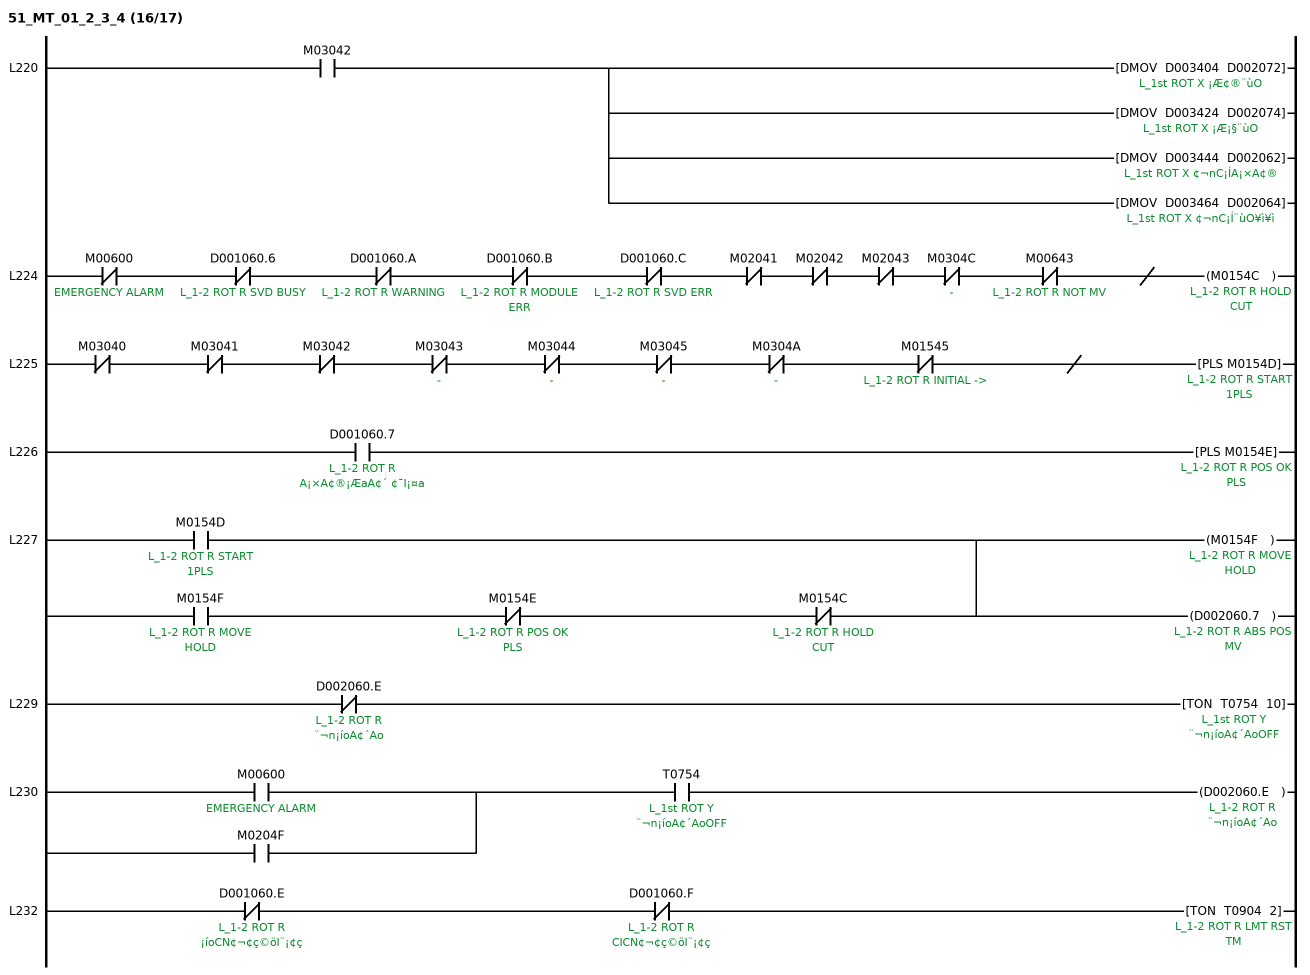
[picture p264: 51_MT_01_2_3_4 rungs L220-L232]
; L220
LOAD      M03042
DMOV      D003404 D002072	// L_1st ROT X ¡Æ¢®¨ùO
DMOV      D003424 D002074	// L_1st ROT X ¡Æ¡§¨ùO
DMOV      D003444 D002062	// L_1st ROT X ¢¬nC¡ÍA¡×A¢®
DMOV      D003464 D002064	// L_1st ROT X ¢¬nC¡Í¨ùO¥ì¥ì
; L224
LOAD NOT  M00600	// EMERGENCY ALARM
AND NOT   D001060.6	// L_1-2 ROT R SVD BUSY
AND NOT   D001060.A	// L_1-2 ROT R WARNING
AND NOT   D001060.B	// L_1-2 ROT R MODULE ERR
AND NOT   D001060.C	// L_1-2 ROT R SVD ERR
AND NOT   M02041
AND NOT   M02042
AND NOT   M02043
AND NOT   M0304C	// -
AND NOT   M00643	// L_1-2 ROT R NOT MV
NOT
OUT       M0154C	// L_1-2 ROT R HOLD CUT
; L225
LOAD NOT  M03040
AND NOT   M03041
AND NOT   M03042
AND NOT   M03043	// -
AND NOT   M03044	// -
AND NOT   M03045	// -
AND NOT   M0304A	// -
AND NOT   M01545	// L_1-2 ROT R INITIAL ->
NOT
OUTP      M0154D	// L_1-2 ROT R START 1PLS
; L226
LOAD      D001060.7	// L_1-2 ROT R A¡×A¢®¡ÆaA¢´ ¢¯I¡¤a
OUTP      M0154E	// L_1-2 ROT R POS OK PLS
; L227
LOAD      M0154D	// L_1-2 ROT R START 1PLS
LOAD      M0154F	// L_1-2 ROT R MOVE HOLD
AND NOT   M0154E	// L_1-2 ROT R POS OK PLS
AND NOT   M0154C	// L_1-2 ROT R HOLD CUT
OR LOAD
OUT       M0154F	// L_1-2 ROT R MOVE HOLD
OUT       D002060.7	// L_1-2 ROT R ABS POS MV
; L229
LOAD NOT  D002060.E	// L_1-2 ROT R ¨¬n¡íoA¢´Ao
TON       T0754 10	// L_1st ROT Y ¨¬n¡íoA¢´AoOFF
; L230
LOAD      M00600	// EMERGENCY ALARM
OR        M0204F
AND       T0754	// L_1st ROT Y ¨¬n¡íoA¢´AoOFF
OUT       D002060.E	// L_1-2 ROT R ¨¬n¡íoA¢´Ao
; L232
LOAD NOT  D001060.E	// L_1-2 ROT R ¡íoCN¢¬¢ç©öI¨¡¢ç
AND NOT   D001060.F	// L_1-2 ROT R CICN¢¬¢ç©öI¨¡¢ç
TON       T0904 2	// L_1-2 ROT R LMT RST TM

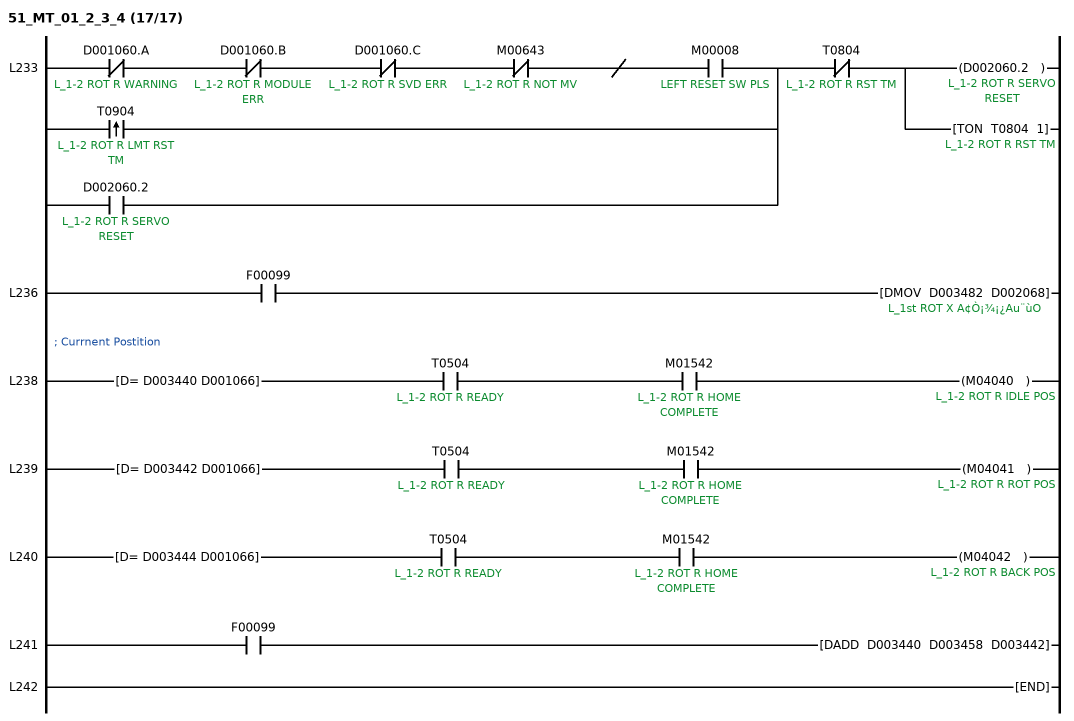
; L233
LOAD NOT  D001060.A	// L_1-2 ROT R WARNING
AND NOT   D001060.B	// L_1-2 ROT R MODULE ERR
AND NOT   D001060.C	// L_1-2 ROT R SVD ERR
AND NOT   M00643	// L_1-2 ROT R NOT MV
NOT
AND       M00008	// LEFT RESET SW PLS
ORP       T0904	// L_1-2 ROT R LMT RST TM
OR        D002060.2	// L_1-2 ROT R SERVO RESET
AND NOT   T0804	// L_1-2 ROT R RST TM
OUT       D002060.2	// L_1-2 ROT R SERVO RESET
TON       T0804 1	// L_1-2 ROT R RST TM
; L236
LOAD      F00099
DMOV      D003482 D002068	// L_1st ROT X A¢Ò¡¾¡¿Au¨ùO
// Currnent Postition
; L238
LOADD=    D003440 D001066
AND       T0504	// L_1-2 ROT R READY
AND       M01542	// L_1-2 ROT R HOME COMPLETE
OUT       M04040	// L_1-2 ROT R IDLE POS
; L239
LOADD=    D003442 D001066
AND       T0504	// L_1-2 ROT R READY
AND       M01542	// L_1-2 ROT R HOME COMPLETE
OUT       M04041	// L_1-2 ROT R ROT POS
; L240
LOADD=    D003444 D001066
AND       T0504	// L_1-2 ROT R READY
AND       M01542	// L_1-2 ROT R HOME COMPLETE
OUT       M04042	// L_1-2 ROT R BACK POS
; L241
LOAD      F00099
DADD      D003440 D003458 D003442
; L242
END

PROGRAM 52_MT_05_6_7_8 (task: ¨ö¨¬A¥ì CA¡¤I¡¾¡¿¡¤¡Í)

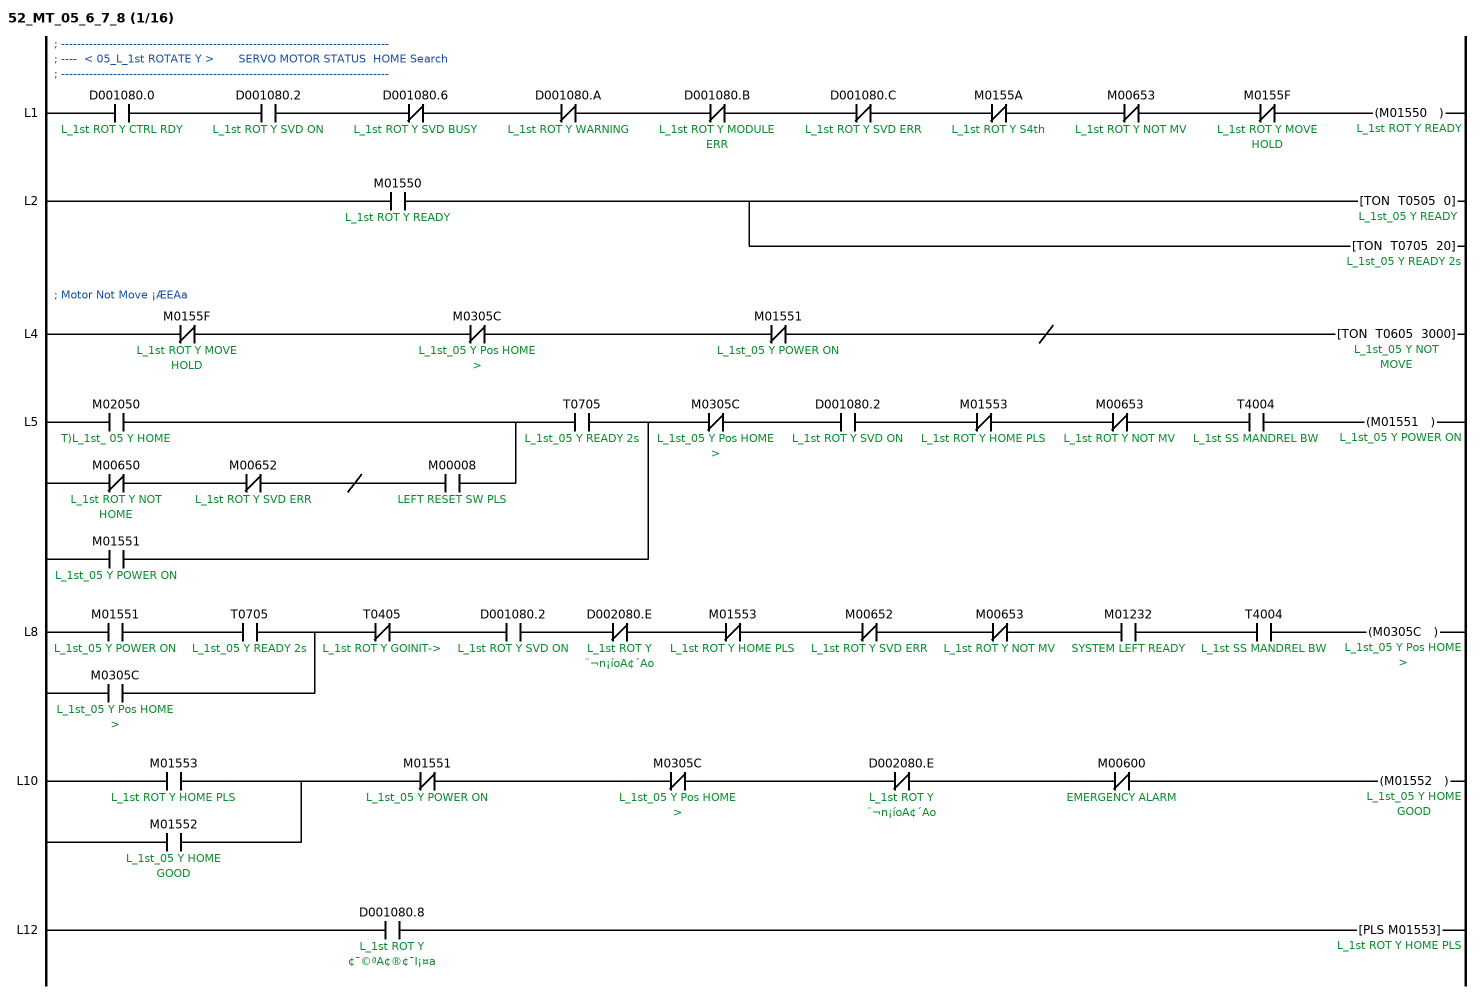
// ----------------------------------------------------------------------------------
// 
// ----  < 05_L_1st ROTATE Y >       SERVO MOTOR STATUS  HOME Search
// 
// ----------------------------------------------------------------------------------
; L1
LOAD      D001080.0	// L_1st ROT Y CTRL RDY
AND       D001080.2	// L_1st ROT Y SVD ON
AND NOT   D001080.6	// L_1st ROT Y SVD BUSY
AND NOT   D001080.A	// L_1st ROT Y WARNING
AND NOT   D001080.B	// L_1st ROT Y MODULE ERR
AND NOT   D001080.C	// L_1st ROT Y SVD ERR
AND NOT   M0155A	// L_1st ROT Y S4th
AND NOT   M00653	// L_1st ROT Y NOT MV
AND NOT   M0155F	// L_1st ROT Y MOVE HOLD
OUT       M01550	// L_1st ROT Y READY
; L2
LOAD      M01550	// L_1st ROT Y READY
TON       T0505 0	// L_1st_05 Y READY
TON       T0705 20	// L_1st_05 Y READY 2s
; L4
LOAD NOT  M0155F	// L_1st ROT Y MOVE HOLD
AND NOT   M0305C	// L_1st_05 Y Pos HOME >
AND NOT   M01551	// L_1st_05 Y POWER ON
NOT
TON       T0605 3000	// L_1st_05 Y NOT MOVE
// output comment: Motor Not Move ¡ÆEAa
; L5
LOAD      M02050	// T)L_1st_ 05 Y HOME
LOAD NOT  M00650	// L_1st ROT Y NOT HOME
AND NOT   M00652	// L_1st ROT Y SVD ERR
NOT
AND       M00008	// LEFT RESET SW PLS
OR LOAD
AND       T0705	// L_1st_05 Y READY 2s
OR        M01551	// L_1st_05 Y POWER ON
AND NOT   M0305C	// L_1st_05 Y Pos HOME >
AND       D001080.2	// L_1st ROT Y SVD ON
AND NOT   M01553	// L_1st ROT Y HOME PLS
AND NOT   M00653	// L_1st ROT Y NOT MV
AND       T4004	// L_1st SS MANDREL BW
OUT       M01551	// L_1st_05 Y POWER ON
; L8
LOAD      M01551	// L_1st_05 Y POWER ON
AND       T0705	// L_1st_05 Y READY 2s
OR        M0305C	// L_1st_05 Y Pos HOME >
AND NOT   T0405	// L_1st ROT Y GOINIT->
AND       D001080.2	// L_1st ROT Y SVD ON
AND NOT   D002080.E	// L_1st ROT Y ¨¬n¡íoA¢´Ao
AND NOT   M01553	// L_1st ROT Y HOME PLS
AND NOT   M00652	// L_1st ROT Y SVD ERR
AND NOT   M00653	// L_1st ROT Y NOT MV
AND       M01232	// SYSTEM LEFT READY
AND       T4004	// L_1st SS MANDREL BW
OUT       M0305C	// L_1st_05 Y Pos HOME >
; L10
LOAD      M01553	// L_1st ROT Y HOME PLS
OR        M01552	// L_1st_05 Y HOME GOOD
AND NOT   M01551	// L_1st_05 Y POWER ON
AND NOT   M0305C	// L_1st_05 Y Pos HOME >
AND NOT   D002080.E	// L_1st ROT Y ¨¬n¡íoA¢´Ao
AND NOT   M00600	// EMERGENCY ALARM
OUT       M01552	// L_1st_05 Y HOME GOOD
; L12
LOAD      D001080.8	// L_1st ROT Y ¢¯©ªA¢®¢¯I¡¤a
OUTP      M01553	// L_1st ROT Y HOME PLS

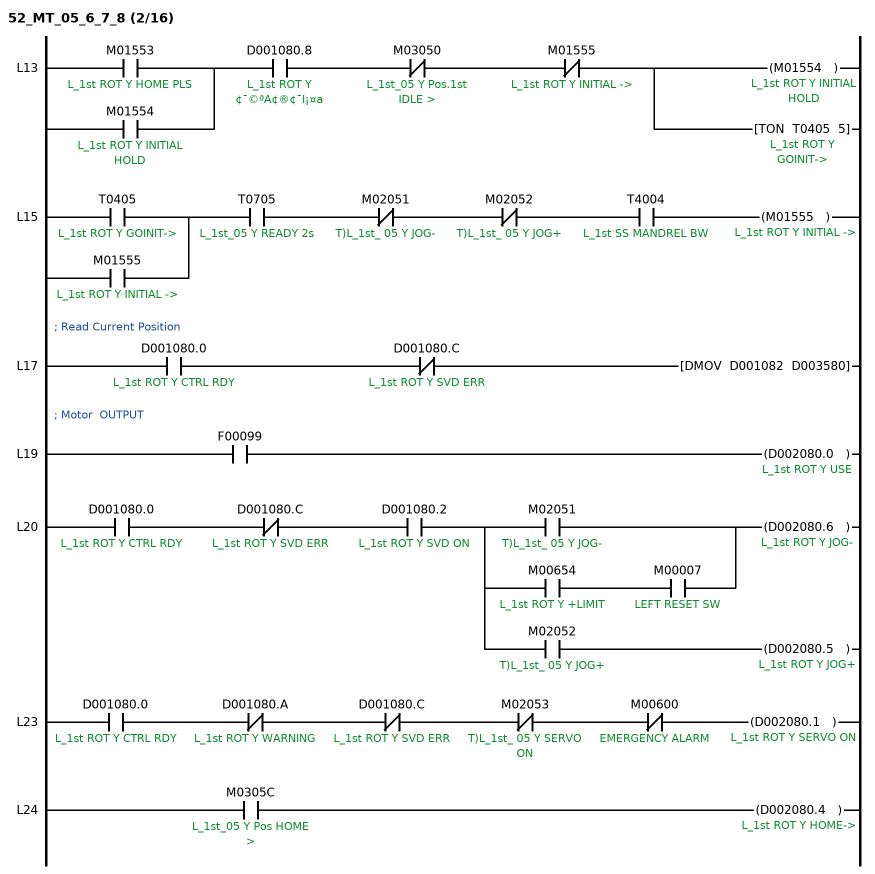
; L13
LOAD      M01553	// L_1st ROT Y HOME PLS
OR        M01554	// L_1st ROT Y INITIAL HOLD
AND       D001080.8	// L_1st ROT Y ¢¯©ªA¢®¢¯I¡¤a
AND NOT   M03050	// L_1st_05 Y Pos.1st IDLE >
AND NOT   M01555	// L_1st ROT Y INITIAL ->
OUT       M01554	// L_1st ROT Y INITIAL HOLD
TON       T0405 5	// L_1st ROT Y GOINIT->
; L15
LOAD      T0405	// L_1st ROT Y GOINIT->
OR        M01555	// L_1st ROT Y INITIAL ->
AND       T0705	// L_1st_05 Y READY 2s
AND NOT   M02051	// T)L_1st_ 05 Y JOG-
AND NOT   M02052	// T)L_1st_ 05 Y JOG+
AND       T4004	// L_1st SS MANDREL BW
OUT       M01555	// L_1st ROT Y INITIAL ->
; L17
LOAD      D001080.0	// L_1st ROT Y CTRL RDY
AND NOT   D001080.C	// L_1st ROT Y SVD ERR
DMOV      D001082 D003580
// output comment: Read Current Position
//  Motor  OUTPUT
; L19
LOAD      F00099
OUT       D002080.0	// L_1st ROT Y USE
; L20
LOAD      D001080.0	// L_1st ROT Y CTRL RDY
AND NOT   D001080.C	// L_1st ROT Y SVD ERR
AND       D001080.2	// L_1st ROT Y SVD ON
MPUSH
LOAD      M02051	// T)L_1st_ 05 Y JOG-
LOAD      M00654	// L_1st ROT Y +LIMIT
AND       M00007	// LEFT RESET SW
OR LOAD
AND LOAD
OUT       D002080.6	// L_1st ROT Y JOG-
MPOP
AND       M02052	// T)L_1st_ 05 Y JOG+
OUT       D002080.5	// L_1st ROT Y JOG+
; L23
LOAD      D001080.0	// L_1st ROT Y CTRL RDY
AND NOT   D001080.A	// L_1st ROT Y WARNING
AND NOT   D001080.C	// L_1st ROT Y SVD ERR
AND NOT   M02053	// T)L_1st_ 05 Y SERVO ON
AND NOT   M00600	// EMERGENCY ALARM
OUT       D002080.1	// L_1st ROT Y SERVO ON
; L24
LOAD      M0305C	// L_1st_05 Y Pos HOME >
OUT       D002080.4	// L_1st ROT Y HOME->

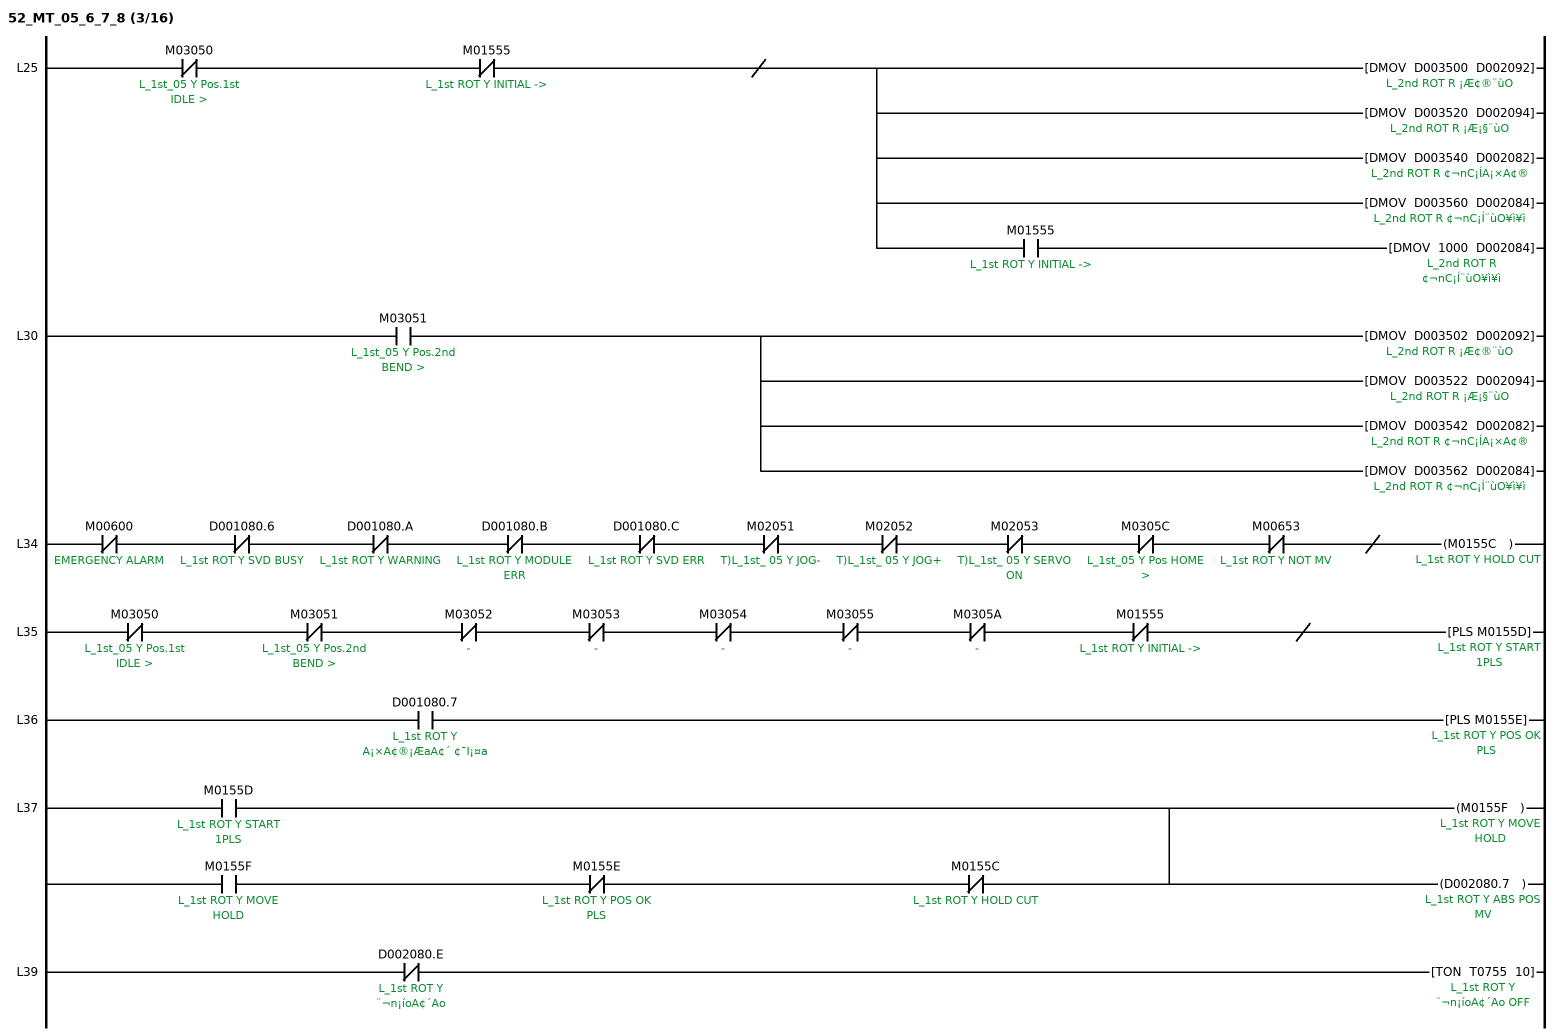
; L25
LOAD NOT  M03050	// L_1st_05 Y Pos.1st IDLE >
AND NOT   M01555	// L_1st ROT Y INITIAL ->
NOT
DMOV      D003500 D002092	// L_2nd ROT R ¡Æ¢®¨ùO
DMOV      D003520 D002094	// L_2nd ROT R ¡Æ¡§¨ùO
DMOV      D003540 D002082	// L_2nd ROT R ¢¬nC¡ÍA¡×A¢®
DMOV      D003560 D002084	// L_2nd ROT R ¢¬nC¡Í¨ùO¥ì¥ì
AND       M01555	// L_1st ROT Y INITIAL ->
DMOV      1000 D002084	// L_2nd ROT R ¢¬nC¡Í¨ùO¥ì¥ì
; L30
LOAD      M03051	// L_1st_05 Y Pos.2nd BEND >
DMOV      D003502 D002092	// L_2nd ROT R ¡Æ¢®¨ùO
DMOV      D003522 D002094	// L_2nd ROT R ¡Æ¡§¨ùO
DMOV      D003542 D002082	// L_2nd ROT R ¢¬nC¡ÍA¡×A¢®
DMOV      D003562 D002084	// L_2nd ROT R ¢¬nC¡Í¨ùO¥ì¥ì
; L34
LOAD NOT  M00600	// EMERGENCY ALARM
AND NOT   D001080.6	// L_1st ROT Y SVD BUSY
AND NOT   D001080.A	// L_1st ROT Y WARNING
AND NOT   D001080.B	// L_1st ROT Y MODULE ERR
AND NOT   D001080.C	// L_1st ROT Y SVD ERR
AND NOT   M02051	// T)L_1st_ 05 Y JOG-
AND NOT   M02052	// T)L_1st_ 05 Y JOG+
AND NOT   M02053	// T)L_1st_ 05 Y SERVO ON
AND NOT   M0305C	// L_1st_05 Y Pos HOME >
AND NOT   M00653	// L_1st ROT Y NOT MV
NOT
OUT       M0155C	// L_1st ROT Y HOLD CUT
; L35
LOAD NOT  M03050	// L_1st_05 Y Pos.1st IDLE >
AND NOT   M03051	// L_1st_05 Y Pos.2nd BEND >
AND NOT   M03052	// -
AND NOT   M03053	// -
AND NOT   M03054	// -
AND NOT   M03055	// -
AND NOT   M0305A	// -
AND NOT   M01555	// L_1st ROT Y INITIAL ->
NOT
OUTP      M0155D	// L_1st ROT Y START 1PLS
; L36
LOAD      D001080.7	// L_1st ROT Y A¡×A¢®¡ÆaA¢´ ¢¯I¡¤a
OUTP      M0155E	// L_1st ROT Y POS OK PLS
; L37
LOAD      M0155D	// L_1st ROT Y START 1PLS
LOAD      M0155F	// L_1st ROT Y MOVE HOLD
AND NOT   M0155E	// L_1st ROT Y POS OK PLS
AND NOT   M0155C	// L_1st ROT Y HOLD CUT
OR LOAD
OUT       M0155F	// L_1st ROT Y MOVE HOLD
OUT       D002080.7	// L_1st ROT Y ABS POS MV
; L39
LOAD NOT  D002080.E	// L_1st ROT Y ¨¬n¡íoA¢´Ao
TON       T0755 10	// L_1st ROT Y ¨¬n¡íoA¢´Ao OFF

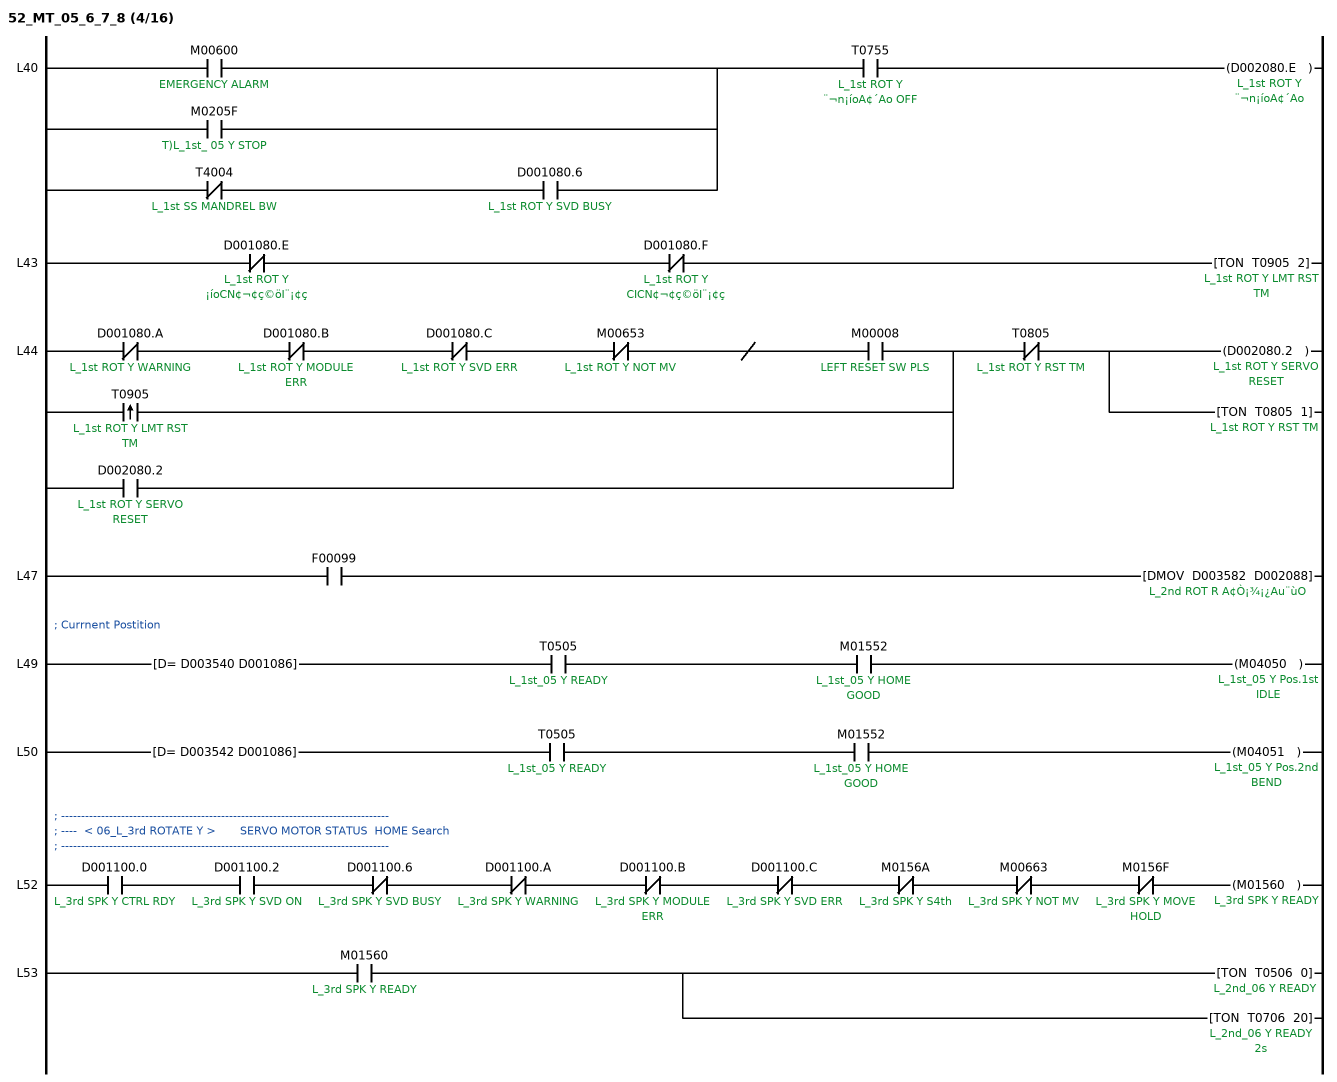
; L40
LOAD      M00600	// EMERGENCY ALARM
OR        M0205F	// T)L_1st_ 05 Y STOP
LOAD NOT  T4004	// L_1st SS MANDREL BW
AND       D001080.6	// L_1st ROT Y SVD BUSY
OR LOAD
AND       T0755	// L_1st ROT Y ¨¬n¡íoA¢´Ao OFF
OUT       D002080.E	// L_1st ROT Y ¨¬n¡íoA¢´Ao
; L43
LOAD NOT  D001080.E	// L_1st ROT Y ¡íoCN¢¬¢ç©öI¨¡¢ç
AND NOT   D001080.F	// L_1st ROT Y CICN¢¬¢ç©öI¨¡¢ç
TON       T0905 2	// L_1st ROT Y LMT RST TM
; L44
LOAD NOT  D001080.A	// L_1st ROT Y WARNING
AND NOT   D001080.B	// L_1st ROT Y MODULE ERR
AND NOT   D001080.C	// L_1st ROT Y SVD ERR
AND NOT   M00653	// L_1st ROT Y NOT MV
NOT
AND       M00008	// LEFT RESET SW PLS
ORP       T0905	// L_1st ROT Y LMT RST TM
OR        D002080.2	// L_1st ROT Y SERVO RESET
AND NOT   T0805	// L_1st ROT Y RST TM
OUT       D002080.2	// L_1st ROT Y SERVO RESET
TON       T0805 1	// L_1st ROT Y RST TM
; L47
LOAD      F00099
DMOV      D003582 D002088	// L_2nd ROT R A¢Ò¡¾¡¿Au¨ùO
// Currnent Postition
; L49
LOADD=    D003540 D001086
AND       T0505	// L_1st_05 Y READY
AND       M01552	// L_1st_05 Y HOME GOOD
OUT       M04050	// L_1st_05 Y Pos.1st IDLE
; L50
LOADD=    D003542 D001086
AND       T0505	// L_1st_05 Y READY
AND       M01552	// L_1st_05 Y HOME GOOD
OUT       M04051	// L_1st_05 Y Pos.2nd BEND
// ----------------------------------------------------------------------------------
// 
// ----  < 06_L_3rd ROTATE Y >       SERVO MOTOR STATUS  HOME Search
// 
// ----------------------------------------------------------------------------------
; L52
LOAD      D001100.0	// L_3rd SPK Y CTRL RDY
AND       D001100.2	// L_3rd SPK Y SVD ON
AND NOT   D001100.6	// L_3rd SPK Y SVD BUSY
AND NOT   D001100.A	// L_3rd SPK Y WARNING
AND NOT   D001100.B	// L_3rd SPK Y MODULE ERR
AND NOT   D001100.C	// L_3rd SPK Y SVD ERR
AND NOT   M0156A	// L_3rd SPK Y S4th
AND NOT   M00663	// L_3rd SPK Y NOT MV
AND NOT   M0156F	// L_3rd SPK Y MOVE HOLD
OUT       M01560	// L_3rd SPK Y READY
; L53
LOAD      M01560	// L_3rd SPK Y READY
TON       T0506 0	// L_2nd_06 Y READY
TON       T0706 20	// L_2nd_06 Y READY 2s

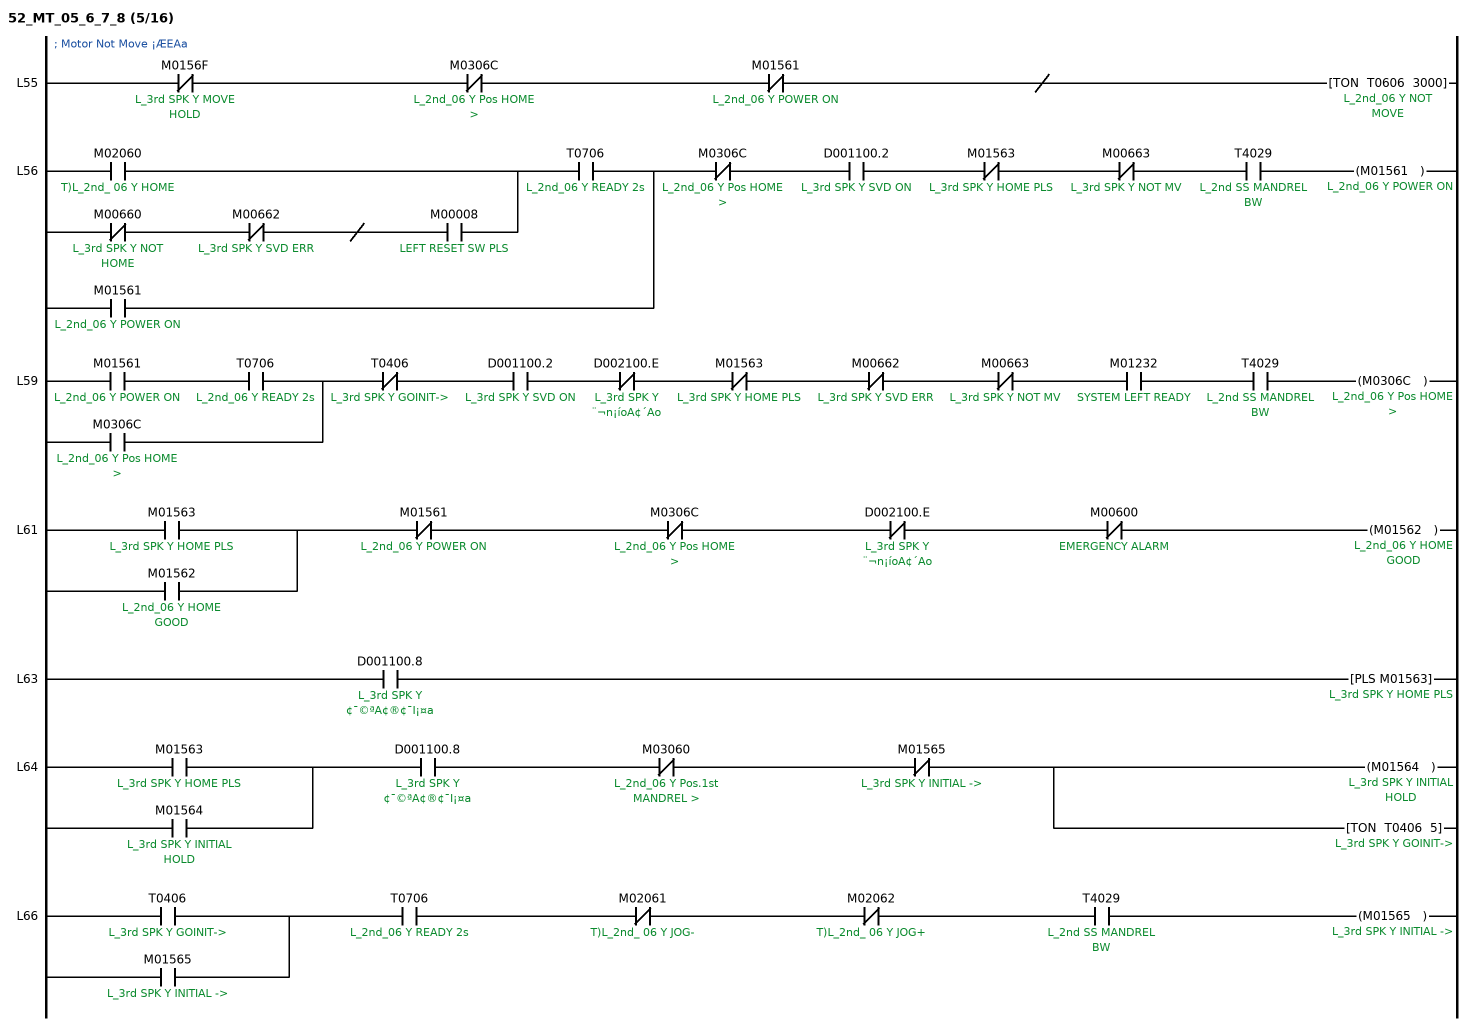
; L55
LOAD NOT  M0156F	// L_3rd SPK Y MOVE HOLD
AND NOT   M0306C	// L_2nd_06 Y Pos HOME >
AND NOT   M01561	// L_2nd_06 Y POWER ON
NOT
TON       T0606 3000	// L_2nd_06 Y NOT MOVE
// output comment: Motor Not Move ¡ÆEAa
; L56
LOAD      M02060	// T)L_2nd_ 06 Y HOME
LOAD NOT  M00660	// L_3rd SPK Y NOT HOME
AND NOT   M00662	// L_3rd SPK Y SVD ERR
NOT
AND       M00008	// LEFT RESET SW PLS
OR LOAD
AND       T0706	// L_2nd_06 Y READY 2s
OR        M01561	// L_2nd_06 Y POWER ON
AND NOT   M0306C	// L_2nd_06 Y Pos HOME >
AND       D001100.2	// L_3rd SPK Y SVD ON
AND NOT   M01563	// L_3rd SPK Y HOME PLS
AND NOT   M00663	// L_3rd SPK Y NOT MV
AND       T4029	// L_2nd SS MANDREL BW
OUT       M01561	// L_2nd_06 Y POWER ON
; L59
LOAD      M01561	// L_2nd_06 Y POWER ON
AND       T0706	// L_2nd_06 Y READY 2s
OR        M0306C	// L_2nd_06 Y Pos HOME >
AND NOT   T0406	// L_3rd SPK Y GOINIT->
AND       D001100.2	// L_3rd SPK Y SVD ON
AND NOT   D002100.E	// L_3rd SPK Y ¨¬n¡íoA¢´Ao
AND NOT   M01563	// L_3rd SPK Y HOME PLS
AND NOT   M00662	// L_3rd SPK Y SVD ERR
AND NOT   M00663	// L_3rd SPK Y NOT MV
AND       M01232	// SYSTEM LEFT READY
AND       T4029	// L_2nd SS MANDREL BW
OUT       M0306C	// L_2nd_06 Y Pos HOME >
; L61
LOAD      M01563	// L_3rd SPK Y HOME PLS
OR        M01562	// L_2nd_06 Y HOME GOOD
AND NOT   M01561	// L_2nd_06 Y POWER ON
AND NOT   M0306C	// L_2nd_06 Y Pos HOME >
AND NOT   D002100.E	// L_3rd SPK Y ¨¬n¡íoA¢´Ao
AND NOT   M00600	// EMERGENCY ALARM
OUT       M01562	// L_2nd_06 Y HOME GOOD
; L63
LOAD      D001100.8	// L_3rd SPK Y ¢¯©ªA¢®¢¯I¡¤a
OUTP      M01563	// L_3rd SPK Y HOME PLS
; L64
LOAD      M01563	// L_3rd SPK Y HOME PLS
OR        M01564	// L_3rd SPK Y INITIAL HOLD
AND       D001100.8	// L_3rd SPK Y ¢¯©ªA¢®¢¯I¡¤a
AND NOT   M03060	// L_2nd_06 Y Pos.1st MANDREL >
AND NOT   M01565	// L_3rd SPK Y INITIAL ->
OUT       M01564	// L_3rd SPK Y INITIAL HOLD
TON       T0406 5	// L_3rd SPK Y GOINIT->
; L66
LOAD      T0406	// L_3rd SPK Y GOINIT->
OR        M01565	// L_3rd SPK Y INITIAL ->
AND       T0706	// L_2nd_06 Y READY 2s
AND NOT   M02061	// T)L_2nd_ 06 Y JOG-
AND NOT   M02062	// T)L_2nd_ 06 Y JOG+
AND       T4029	// L_2nd SS MANDREL BW
OUT       M01565	// L_3rd SPK Y INITIAL ->

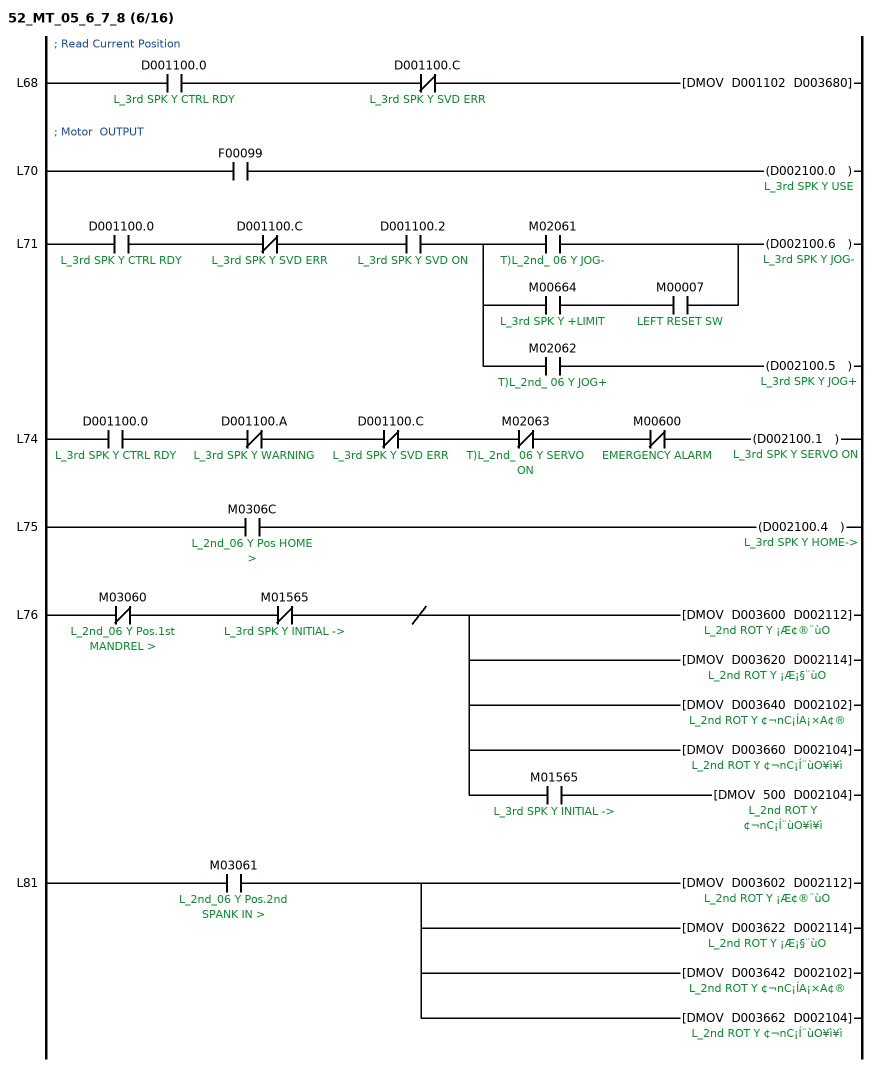
; L68
LOAD      D001100.0	// L_3rd SPK Y CTRL RDY
AND NOT   D001100.C	// L_3rd SPK Y SVD ERR
DMOV      D001102 D003680
// output comment: Read Current Position
//  Motor  OUTPUT
; L70
LOAD      F00099
OUT       D002100.0	// L_3rd SPK Y USE
; L71
LOAD      D001100.0	// L_3rd SPK Y CTRL RDY
AND NOT   D001100.C	// L_3rd SPK Y SVD ERR
AND       D001100.2	// L_3rd SPK Y SVD ON
MPUSH
LOAD      M02061	// T)L_2nd_ 06 Y JOG-
LOAD      M00664	// L_3rd SPK Y +LIMIT
AND       M00007	// LEFT RESET SW
OR LOAD
AND LOAD
OUT       D002100.6	// L_3rd SPK Y JOG-
MPOP
AND       M02062	// T)L_2nd_ 06 Y JOG+
OUT       D002100.5	// L_3rd SPK Y JOG+
; L74
LOAD      D001100.0	// L_3rd SPK Y CTRL RDY
AND NOT   D001100.A	// L_3rd SPK Y WARNING
AND NOT   D001100.C	// L_3rd SPK Y SVD ERR
AND NOT   M02063	// T)L_2nd_ 06 Y SERVO ON
AND NOT   M00600	// EMERGENCY ALARM
OUT       D002100.1	// L_3rd SPK Y SERVO ON
; L75
LOAD      M0306C	// L_2nd_06 Y Pos HOME >
OUT       D002100.4	// L_3rd SPK Y HOME->
; L76
LOAD NOT  M03060	// L_2nd_06 Y Pos.1st MANDREL >
AND NOT   M01565	// L_3rd SPK Y INITIAL ->
NOT
DMOV      D003600 D002112	// L_2nd ROT Y ¡Æ¢®¨ùO
DMOV      D003620 D002114	// L_2nd ROT Y ¡Æ¡§¨ùO
DMOV      D003640 D002102	// L_2nd ROT Y ¢¬nC¡ÍA¡×A¢®
DMOV      D003660 D002104	// L_2nd ROT Y ¢¬nC¡Í¨ùO¥ì¥ì
AND       M01565	// L_3rd SPK Y INITIAL ->
DMOV      500 D002104	// L_2nd ROT Y ¢¬nC¡Í¨ùO¥ì¥ì
; L81
LOAD      M03061	// L_2nd_06 Y Pos.2nd SPANK IN >
DMOV      D003602 D002112	// L_2nd ROT Y ¡Æ¢®¨ùO
DMOV      D003622 D002114	// L_2nd ROT Y ¡Æ¡§¨ùO
DMOV      D003642 D002102	// L_2nd ROT Y ¢¬nC¡ÍA¡×A¢®
DMOV      D003662 D002104	// L_2nd ROT Y ¢¬nC¡Í¨ùO¥ì¥ì

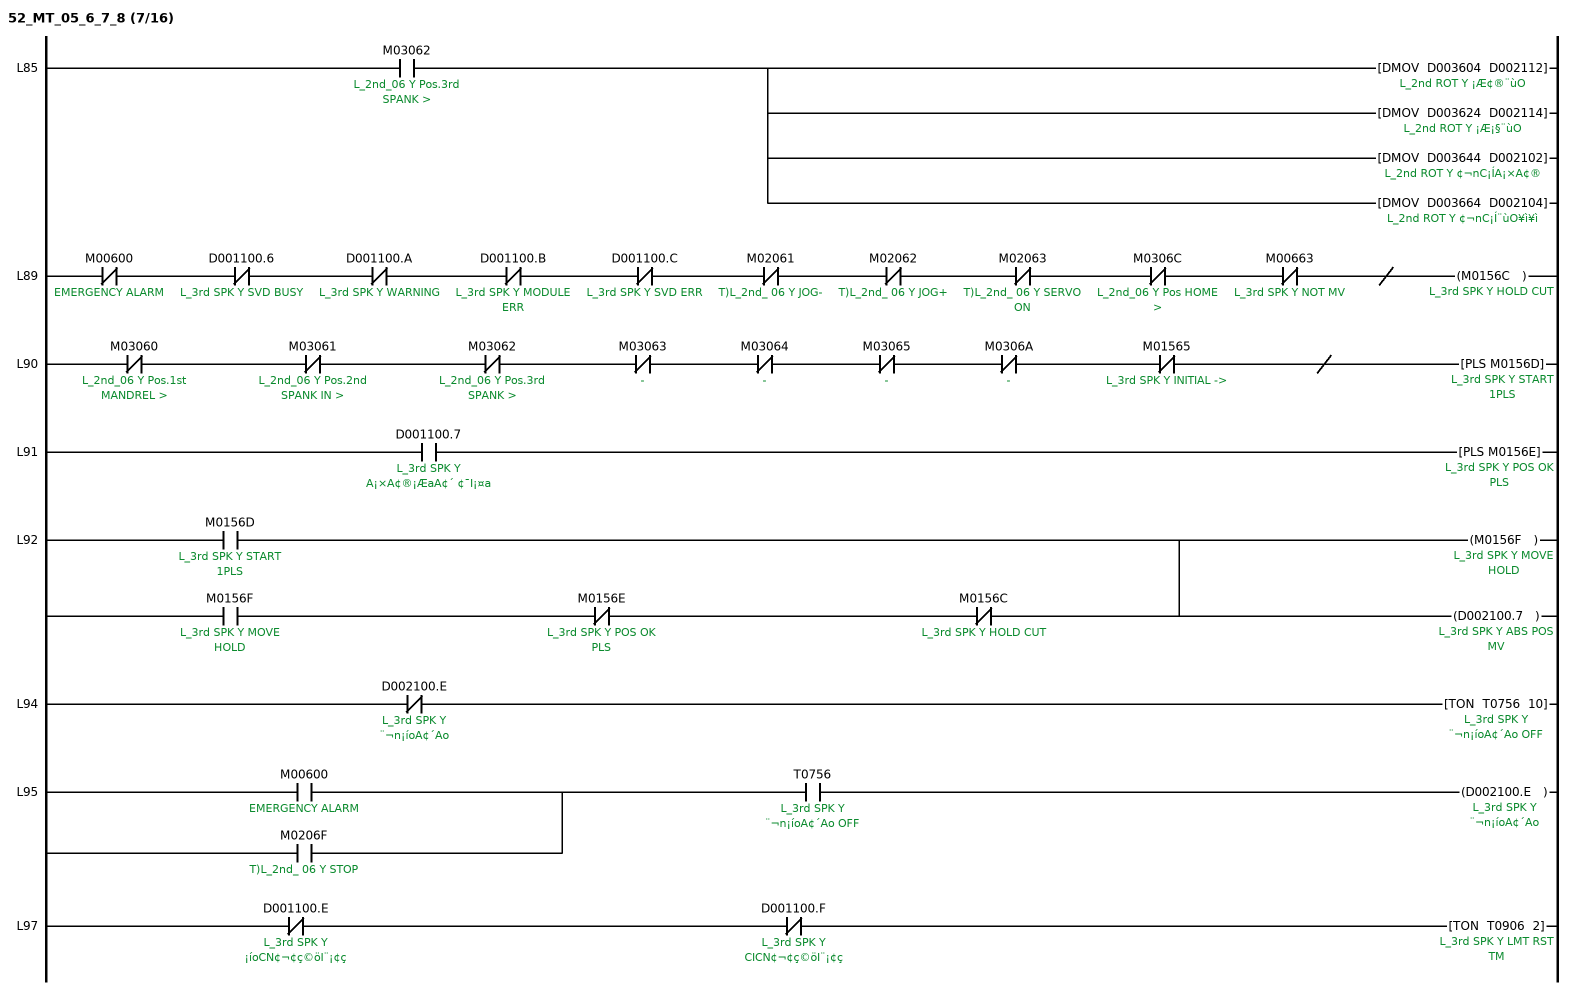
; L85
LOAD      M03062	// L_2nd_06 Y Pos.3rd SPANK >
DMOV      D003604 D002112	// L_2nd ROT Y ¡Æ¢®¨ùO
DMOV      D003624 D002114	// L_2nd ROT Y ¡Æ¡§¨ùO
DMOV      D003644 D002102	// L_2nd ROT Y ¢¬nC¡ÍA¡×A¢®
DMOV      D003664 D002104	// L_2nd ROT Y ¢¬nC¡Í¨ùO¥ì¥ì
; L89
LOAD NOT  M00600	// EMERGENCY ALARM
AND NOT   D001100.6	// L_3rd SPK Y SVD BUSY
AND NOT   D001100.A	// L_3rd SPK Y WARNING
AND NOT   D001100.B	// L_3rd SPK Y MODULE ERR
AND NOT   D001100.C	// L_3rd SPK Y SVD ERR
AND NOT   M02061	// T)L_2nd_ 06 Y JOG-
AND NOT   M02062	// T)L_2nd_ 06 Y JOG+
AND NOT   M02063	// T)L_2nd_ 06 Y SERVO ON
AND NOT   M0306C	// L_2nd_06 Y Pos HOME >
AND NOT   M00663	// L_3rd SPK Y NOT MV
NOT
OUT       M0156C	// L_3rd SPK Y HOLD CUT
; L90
LOAD NOT  M03060	// L_2nd_06 Y Pos.1st MANDREL >
AND NOT   M03061	// L_2nd_06 Y Pos.2nd SPANK IN >
AND NOT   M03062	// L_2nd_06 Y Pos.3rd SPANK >
AND NOT   M03063	// -
AND NOT   M03064	// -
AND NOT   M03065	// -
AND NOT   M0306A	// -
AND NOT   M01565	// L_3rd SPK Y INITIAL ->
NOT
OUTP      M0156D	// L_3rd SPK Y START 1PLS
; L91
LOAD      D001100.7	// L_3rd SPK Y A¡×A¢®¡ÆaA¢´ ¢¯I¡¤a
OUTP      M0156E	// L_3rd SPK Y POS OK PLS
; L92
LOAD      M0156D	// L_3rd SPK Y START 1PLS
LOAD      M0156F	// L_3rd SPK Y MOVE HOLD
AND NOT   M0156E	// L_3rd SPK Y POS OK PLS
AND NOT   M0156C	// L_3rd SPK Y HOLD CUT
OR LOAD
OUT       M0156F	// L_3rd SPK Y MOVE HOLD
OUT       D002100.7	// L_3rd SPK Y ABS POS MV
; L94
LOAD NOT  D002100.E	// L_3rd SPK Y ¨¬n¡íoA¢´Ao
TON       T0756 10	// L_3rd SPK Y ¨¬n¡íoA¢´Ao OFF
; L95
LOAD      M00600	// EMERGENCY ALARM
OR        M0206F	// T)L_2nd_ 06 Y STOP
AND       T0756	// L_3rd SPK Y ¨¬n¡íoA¢´Ao OFF
OUT       D002100.E	// L_3rd SPK Y ¨¬n¡íoA¢´Ao
; L97
LOAD NOT  D001100.E	// L_3rd SPK Y ¡íoCN¢¬¢ç©öI¨¡¢ç
AND NOT   D001100.F	// L_3rd SPK Y CICN¢¬¢ç©öI¨¡¢ç
TON       T0906 2	// L_3rd SPK Y LMT RST TM

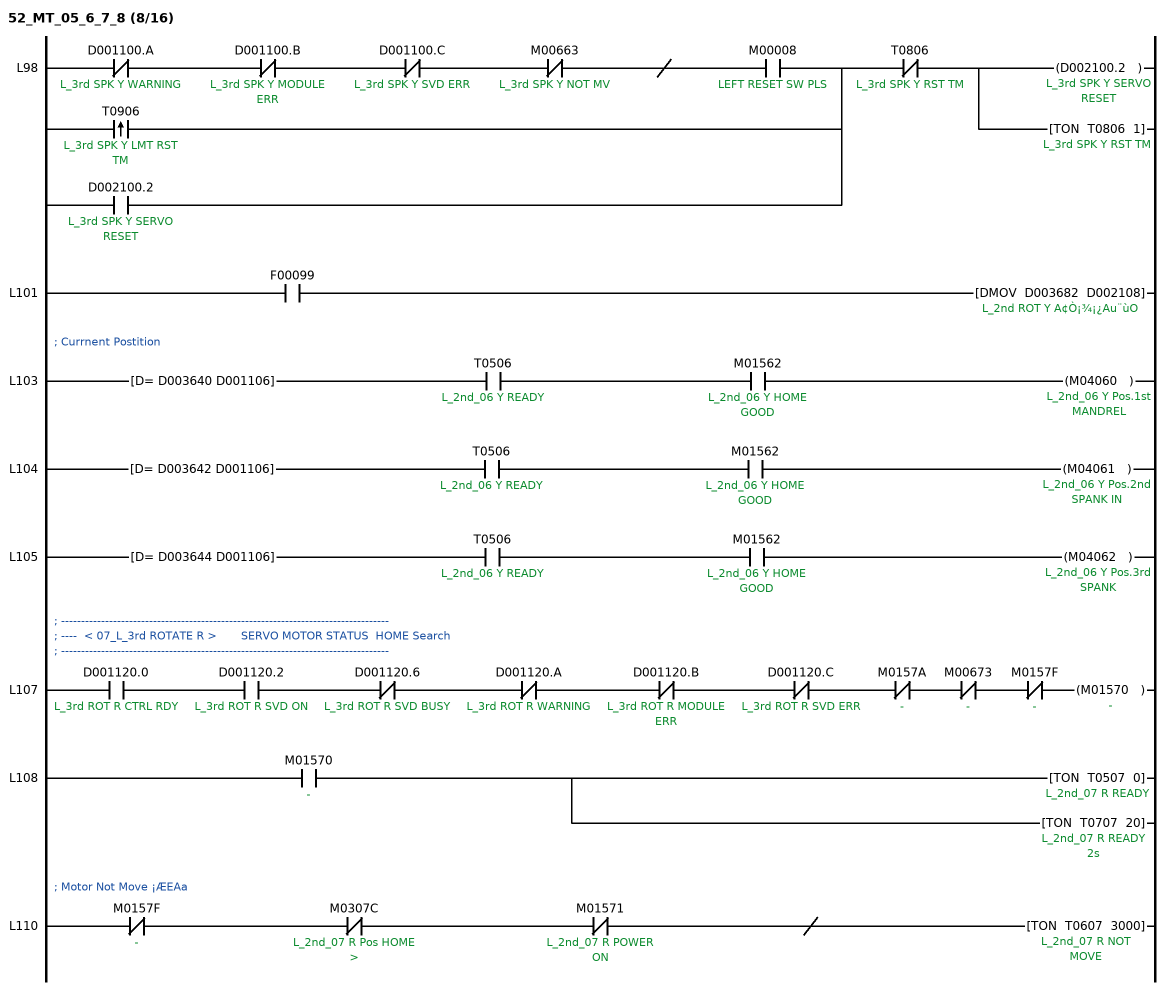
; L98
LOAD NOT  D001100.A	// L_3rd SPK Y WARNING
AND NOT   D001100.B	// L_3rd SPK Y MODULE ERR
AND NOT   D001100.C	// L_3rd SPK Y SVD ERR
AND NOT   M00663	// L_3rd SPK Y NOT MV
NOT
AND       M00008	// LEFT RESET SW PLS
ORP       T0906	// L_3rd SPK Y LMT RST TM
OR        D002100.2	// L_3rd SPK Y SERVO RESET
AND NOT   T0806	// L_3rd SPK Y RST TM
OUT       D002100.2	// L_3rd SPK Y SERVO RESET
TON       T0806 1	// L_3rd SPK Y RST TM
; L101
LOAD      F00099
DMOV      D003682 D002108	// L_2nd ROT Y A¢Ò¡¾¡¿Au¨ùO
// Currnent Postition
; L103
LOADD=    D003640 D001106
AND       T0506	// L_2nd_06 Y READY
AND       M01562	// L_2nd_06 Y HOME GOOD
OUT       M04060	// L_2nd_06 Y Pos.1st MANDREL
; L104
LOADD=    D003642 D001106
AND       T0506	// L_2nd_06 Y READY
AND       M01562	// L_2nd_06 Y HOME GOOD
OUT       M04061	// L_2nd_06 Y Pos.2nd SPANK IN
; L105
LOADD=    D003644 D001106
AND       T0506	// L_2nd_06 Y READY
AND       M01562	// L_2nd_06 Y HOME GOOD
OUT       M04062	// L_2nd_06 Y Pos.3rd SPANK
// ----------------------------------------------------------------------------------
// 
// ----  < 07_L_3rd ROTATE R >       SERVO MOTOR STATUS  HOME Search
// 
// ----------------------------------------------------------------------------------
; L107
LOAD      D001120.0	// L_3rd ROT R CTRL RDY
AND       D001120.2	// L_3rd ROT R SVD ON
AND NOT   D001120.6	// L_3rd ROT R SVD BUSY
AND NOT   D001120.A	// L_3rd ROT R WARNING
AND NOT   D001120.B	// L_3rd ROT R MODULE ERR
AND NOT   D001120.C	// L_3rd ROT R SVD ERR
AND NOT   M0157A	// -
AND NOT   M00673	// -
AND NOT   M0157F	// -
OUT       M01570	// -
; L108
LOAD      M01570	// -
TON       T0507 0	// L_2nd_07 R READY
TON       T0707 20	// L_2nd_07 R READY 2s
; L110
LOAD NOT  M0157F	// -
AND NOT   M0307C	// L_2nd_07 R Pos HOME >
AND NOT   M01571	// L_2nd_07 R POWER ON
NOT
TON       T0607 3000	// L_2nd_07 R NOT MOVE
// output comment: Motor Not Move ¡ÆEAa

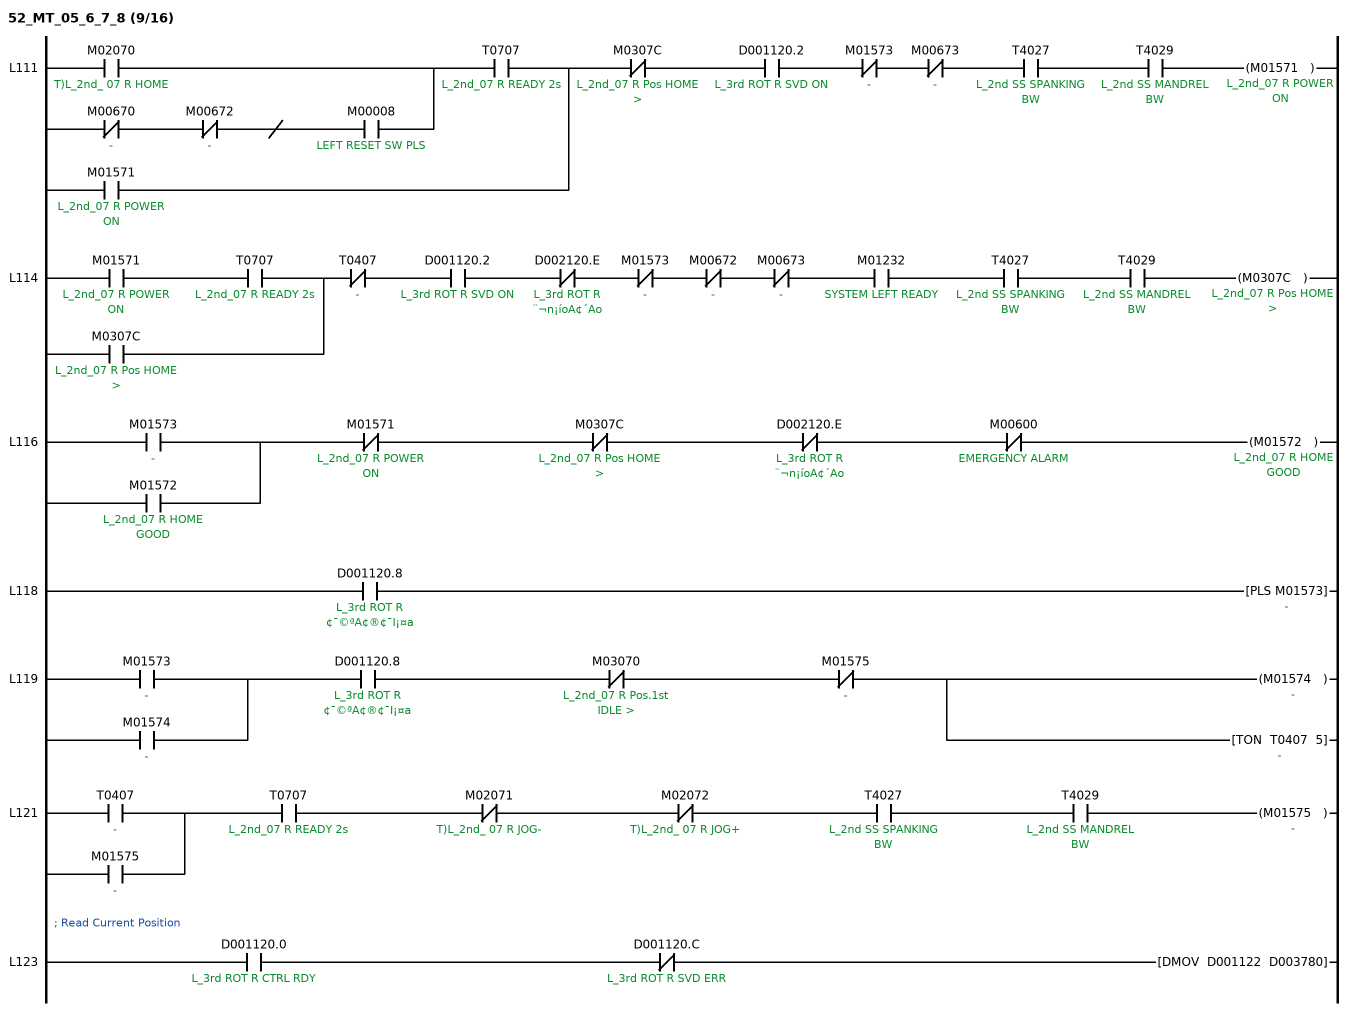
; L111
LOAD      M02070	// T)L_2nd_ 07 R HOME
LOAD NOT  M00670	// -
AND NOT   M00672	// -
NOT
AND       M00008	// LEFT RESET SW PLS
OR LOAD
AND       T0707	// L_2nd_07 R READY 2s
OR        M01571	// L_2nd_07 R POWER ON
AND NOT   M0307C	// L_2nd_07 R Pos HOME >
AND       D001120.2	// L_3rd ROT R SVD ON
AND NOT   M01573	// -
AND NOT   M00673	// -
AND       T4027	// L_2nd SS SPANKING BW
AND       T4029	// L_2nd SS MANDREL BW
OUT       M01571	// L_2nd_07 R POWER ON
; L114
LOAD      M01571	// L_2nd_07 R POWER ON
AND       T0707	// L_2nd_07 R READY 2s
OR        M0307C	// L_2nd_07 R Pos HOME >
AND NOT   T0407	// -
AND       D001120.2	// L_3rd ROT R SVD ON
AND NOT   D002120.E	// L_3rd ROT R ¨¬n¡íoA¢´Ao
AND NOT   M01573	// -
AND NOT   M00672	// -
AND NOT   M00673	// -
AND       M01232	// SYSTEM LEFT READY
AND       T4027	// L_2nd SS SPANKING BW
AND       T4029	// L_2nd SS MANDREL BW
OUT       M0307C	// L_2nd_07 R Pos HOME >
; L116
LOAD      M01573	// -
OR        M01572	// L_2nd_07 R HOME GOOD
AND NOT   M01571	// L_2nd_07 R POWER ON
AND NOT   M0307C	// L_2nd_07 R Pos HOME >
AND NOT   D002120.E	// L_3rd ROT R ¨¬n¡íoA¢´Ao
AND NOT   M00600	// EMERGENCY ALARM
OUT       M01572	// L_2nd_07 R HOME GOOD
; L118
LOAD      D001120.8	// L_3rd ROT R ¢¯©ªA¢®¢¯I¡¤a
OUTP      M01573	// -
; L119
LOAD      M01573	// -
OR        M01574	// -
AND       D001120.8	// L_3rd ROT R ¢¯©ªA¢®¢¯I¡¤a
AND NOT   M03070	// L_2nd_07 R Pos.1st IDLE >
AND NOT   M01575	// -
OUT       M01574	// -
TON       T0407 5	// -
; L121
LOAD      T0407	// -
OR        M01575	// -
AND       T0707	// L_2nd_07 R READY 2s
AND NOT   M02071	// T)L_2nd_ 07 R JOG-
AND NOT   M02072	// T)L_2nd_ 07 R JOG+
AND       T4027	// L_2nd SS SPANKING BW
AND       T4029	// L_2nd SS MANDREL BW
OUT       M01575	// -
; L123
LOAD      D001120.0	// L_3rd ROT R CTRL RDY
AND NOT   D001120.C	// L_3rd ROT R SVD ERR
DMOV      D001122 D003780
// output comment: Read Current Position

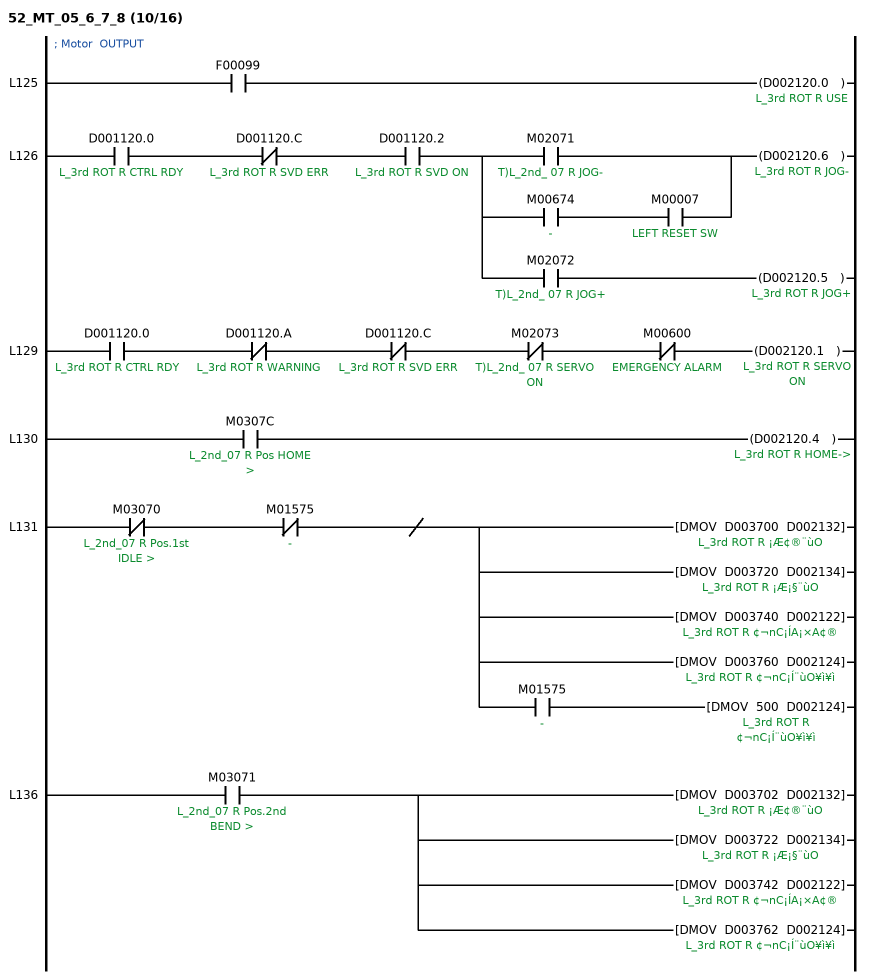
//  Motor  OUTPUT
; L125
LOAD      F00099
OUT       D002120.0	// L_3rd ROT R USE
; L126
LOAD      D001120.0	// L_3rd ROT R CTRL RDY
AND NOT   D001120.C	// L_3rd ROT R SVD ERR
AND       D001120.2	// L_3rd ROT R SVD ON
MPUSH
LOAD      M02071	// T)L_2nd_ 07 R JOG-
LOAD      M00674	// -
AND       M00007	// LEFT RESET SW
OR LOAD
AND LOAD
OUT       D002120.6	// L_3rd ROT R JOG-
MPOP
AND       M02072	// T)L_2nd_ 07 R JOG+
OUT       D002120.5	// L_3rd ROT R JOG+
; L129
LOAD      D001120.0	// L_3rd ROT R CTRL RDY
AND NOT   D001120.A	// L_3rd ROT R WARNING
AND NOT   D001120.C	// L_3rd ROT R SVD ERR
AND NOT   M02073	// T)L_2nd_ 07 R SERVO ON
AND NOT   M00600	// EMERGENCY ALARM
OUT       D002120.1	// L_3rd ROT R SERVO ON
; L130
LOAD      M0307C	// L_2nd_07 R Pos HOME >
OUT       D002120.4	// L_3rd ROT R HOME->
; L131
LOAD NOT  M03070	// L_2nd_07 R Pos.1st IDLE >
AND NOT   M01575	// -
NOT
DMOV      D003700 D002132	// L_3rd ROT R ¡Æ¢®¨ùO
DMOV      D003720 D002134	// L_3rd ROT R ¡Æ¡§¨ùO
DMOV      D003740 D002122	// L_3rd ROT R ¢¬nC¡ÍA¡×A¢®
DMOV      D003760 D002124	// L_3rd ROT R ¢¬nC¡Í¨ùO¥ì¥ì
AND       M01575	// -
DMOV      500 D002124	// L_3rd ROT R ¢¬nC¡Í¨ùO¥ì¥ì
; L136
LOAD      M03071	// L_2nd_07 R Pos.2nd BEND >
DMOV      D003702 D002132	// L_3rd ROT R ¡Æ¢®¨ùO
DMOV      D003722 D002134	// L_3rd ROT R ¡Æ¡§¨ùO
DMOV      D003742 D002122	// L_3rd ROT R ¢¬nC¡ÍA¡×A¢®
DMOV      D003762 D002124	// L_3rd ROT R ¢¬nC¡Í¨ùO¥ì¥ì

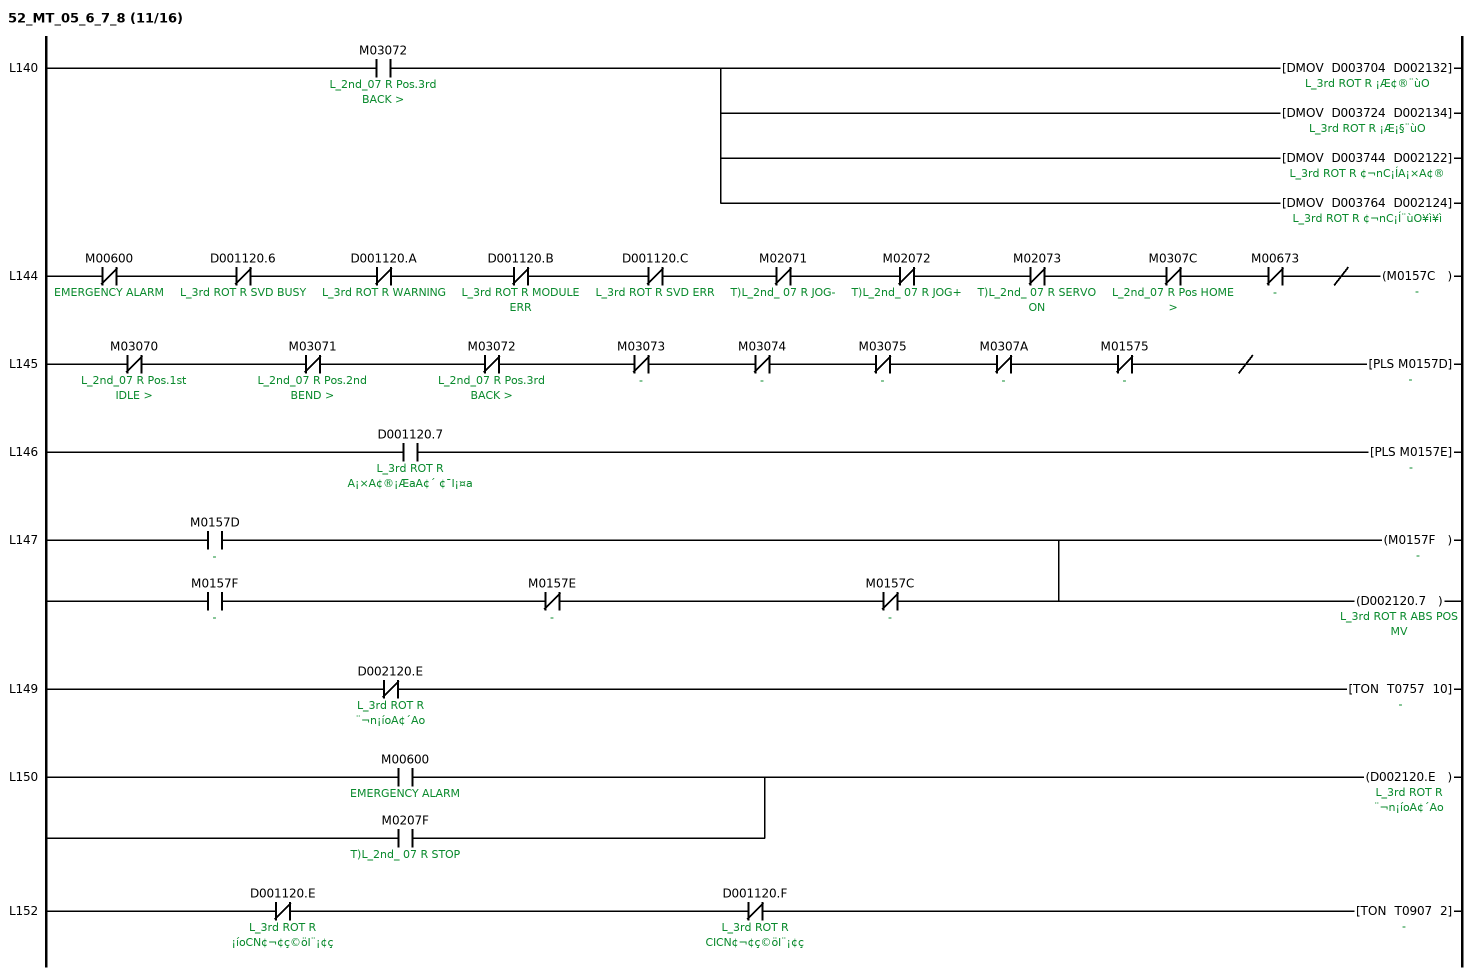
; L140
LOAD      M03072	// L_2nd_07 R Pos.3rd BACK >
DMOV      D003704 D002132	// L_3rd ROT R ¡Æ¢®¨ùO
DMOV      D003724 D002134	// L_3rd ROT R ¡Æ¡§¨ùO
DMOV      D003744 D002122	// L_3rd ROT R ¢¬nC¡ÍA¡×A¢®
DMOV      D003764 D002124	// L_3rd ROT R ¢¬nC¡Í¨ùO¥ì¥ì
; L144
LOAD NOT  M00600	// EMERGENCY ALARM
AND NOT   D001120.6	// L_3rd ROT R SVD BUSY
AND NOT   D001120.A	// L_3rd ROT R WARNING
AND NOT   D001120.B	// L_3rd ROT R MODULE ERR
AND NOT   D001120.C	// L_3rd ROT R SVD ERR
AND NOT   M02071	// T)L_2nd_ 07 R JOG-
AND NOT   M02072	// T)L_2nd_ 07 R JOG+
AND NOT   M02073	// T)L_2nd_ 07 R SERVO ON
AND NOT   M0307C	// L_2nd_07 R Pos HOME >
AND NOT   M00673	// -
NOT
OUT       M0157C	// -
; L145
LOAD NOT  M03070	// L_2nd_07 R Pos.1st IDLE >
AND NOT   M03071	// L_2nd_07 R Pos.2nd BEND >
AND NOT   M03072	// L_2nd_07 R Pos.3rd BACK >
AND NOT   M03073	// -
AND NOT   M03074	// -
AND NOT   M03075	// -
AND NOT   M0307A	// -
AND NOT   M01575	// -
NOT
OUTP      M0157D	// -
; L146
LOAD      D001120.7	// L_3rd ROT R A¡×A¢®¡ÆaA¢´ ¢¯I¡¤a
OUTP      M0157E	// -
; L147
LOAD      M0157D	// -
LOAD      M0157F	// -
AND NOT   M0157E	// -
AND NOT   M0157C	// -
OR LOAD
OUT       M0157F	// -
OUT       D002120.7	// L_3rd ROT R ABS POS MV
; L149
LOAD NOT  D002120.E	// L_3rd ROT R ¨¬n¡íoA¢´Ao
TON       T0757 10	// -
; L150
LOAD      M00600	// EMERGENCY ALARM
OR        M0207F	// T)L_2nd_ 07 R STOP
OUT       D002120.E	// L_3rd ROT R ¨¬n¡íoA¢´Ao
; L152
LOAD NOT  D001120.E	// L_3rd ROT R ¡íoCN¢¬¢ç©öI¨¡¢ç
AND NOT   D001120.F	// L_3rd ROT R CICN¢¬¢ç©öI¨¡¢ç
TON       T0907 2	// -

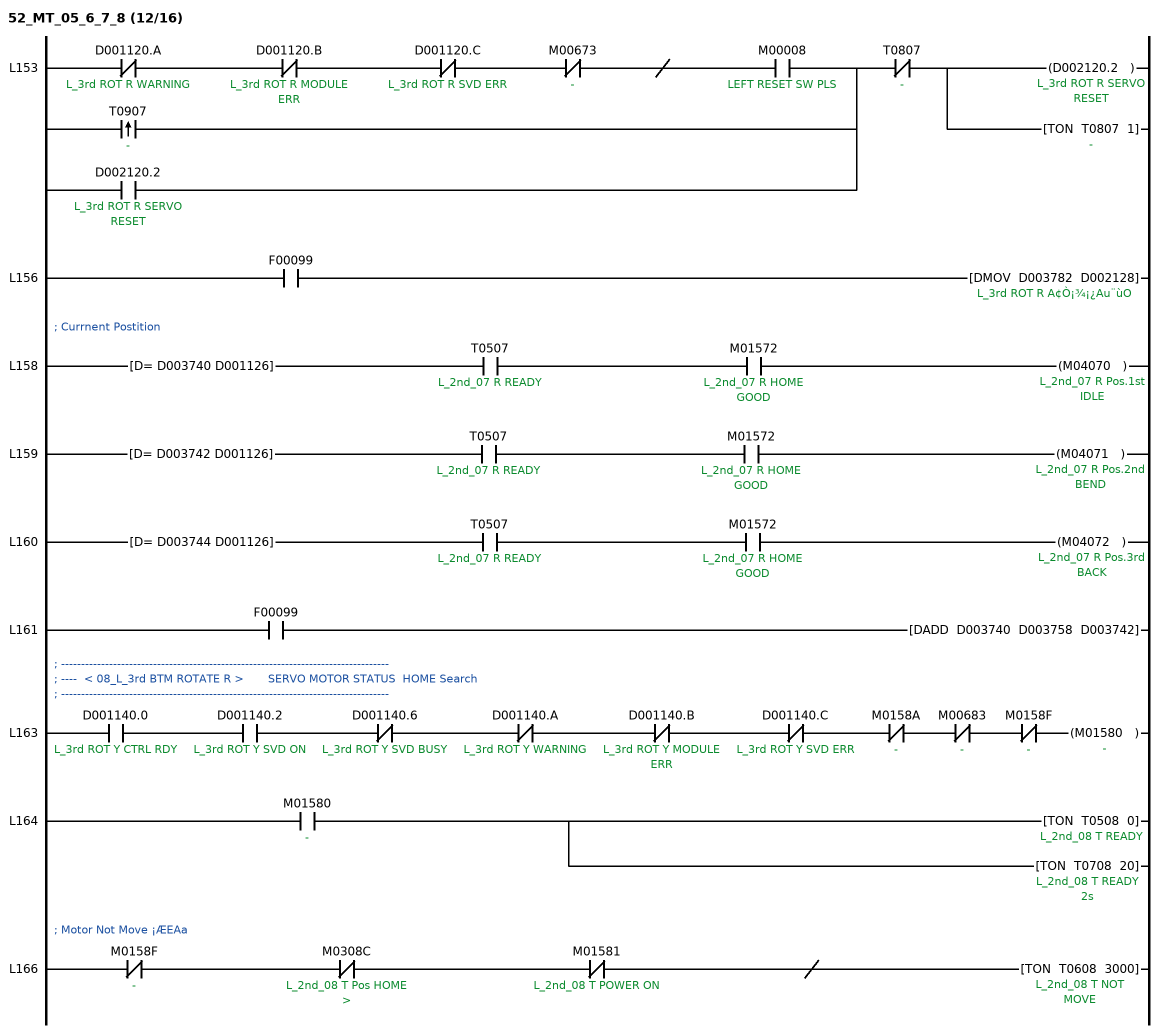
; L153
LOAD NOT  D001120.A	// L_3rd ROT R WARNING
AND NOT   D001120.B	// L_3rd ROT R MODULE ERR
AND NOT   D001120.C	// L_3rd ROT R SVD ERR
AND NOT   M00673	// -
NOT
AND       M00008	// LEFT RESET SW PLS
ORP       T0907	// -
OR        D002120.2	// L_3rd ROT R SERVO RESET
AND NOT   T0807	// -
OUT       D002120.2	// L_3rd ROT R SERVO RESET
TON       T0807 1	// -
; L156
LOAD      F00099
DMOV      D003782 D002128	// L_3rd ROT R A¢Ò¡¾¡¿Au¨ùO
// Currnent Postition
; L158
LOADD=    D003740 D001126
AND       T0507	// L_2nd_07 R READY
AND       M01572	// L_2nd_07 R HOME GOOD
OUT       M04070	// L_2nd_07 R Pos.1st IDLE
; L159
LOADD=    D003742 D001126
AND       T0507	// L_2nd_07 R READY
AND       M01572	// L_2nd_07 R HOME GOOD
OUT       M04071	// L_2nd_07 R Pos.2nd BEND
; L160
LOADD=    D003744 D001126
AND       T0507	// L_2nd_07 R READY
AND       M01572	// L_2nd_07 R HOME GOOD
OUT       M04072	// L_2nd_07 R Pos.3rd BACK
; L161
LOAD      F00099
DADD      D003740 D003758 D003742
// ----------------------------------------------------------------------------------
// 
// ----  < 08_L_3rd BTM ROTATE R >       SERVO MOTOR STATUS  HOME Search
// 
// ----------------------------------------------------------------------------------
; L163
LOAD      D001140.0	// L_3rd ROT Y CTRL RDY
AND       D001140.2	// L_3rd ROT Y SVD ON
AND NOT   D001140.6	// L_3rd ROT Y SVD BUSY
AND NOT   D001140.A	// L_3rd ROT Y WARNING
AND NOT   D001140.B	// L_3rd ROT Y MODULE ERR
AND NOT   D001140.C	// L_3rd ROT Y SVD ERR
AND NOT   M0158A	// -
AND NOT   M00683	// -
AND NOT   M0158F	// -
OUT       M01580	// -
; L164
LOAD      M01580	// -
TON       T0508 0	// L_2nd_08 T READY
TON       T0708 20	// L_2nd_08 T READY 2s
; L166
LOAD NOT  M0158F	// -
AND NOT   M0308C	// L_2nd_08 T Pos HOME >
AND NOT   M01581	// L_2nd_08 T POWER ON
NOT
TON       T0608 3000	// L_2nd_08 T NOT MOVE
// output comment: Motor Not Move ¡ÆEAa

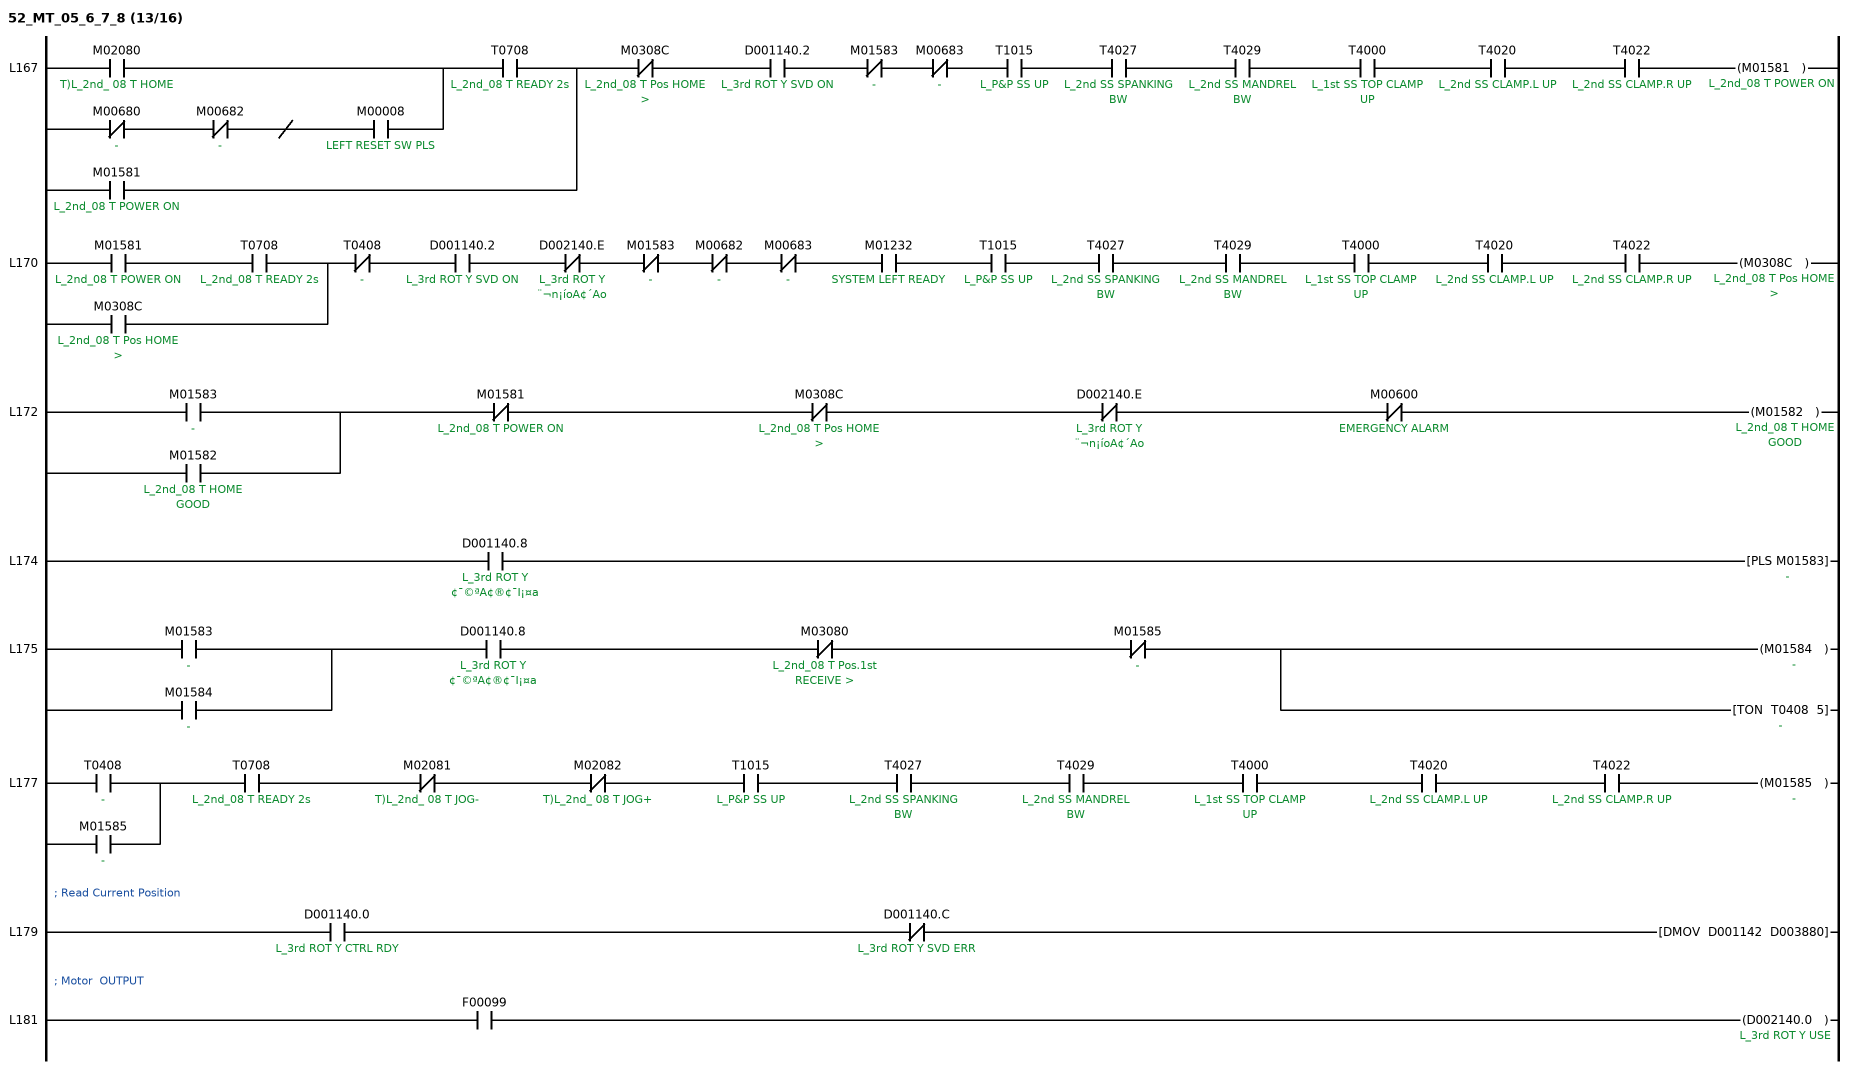
; L167
LOAD      M02080	// T)L_2nd_ 08 T HOME
LOAD NOT  M00680	// -
AND NOT   M00682	// -
NOT
AND       M00008	// LEFT RESET SW PLS
OR LOAD
AND       T0708	// L_2nd_08 T READY 2s
OR        M01581	// L_2nd_08 T POWER ON
AND NOT   M0308C	// L_2nd_08 T Pos HOME >
AND       D001140.2	// L_3rd ROT Y SVD ON
AND NOT   M01583	// -
AND NOT   M00683	// -
AND       T1015	// L_P&P SS UP
AND       T4027	// L_2nd SS SPANKING BW
AND       T4029	// L_2nd SS MANDREL BW
AND       T4000	// L_1st SS TOP CLAMP    UP
AND       T4020	// L_2nd SS CLAMP.L UP
AND       T4022	// L_2nd SS CLAMP.R UP
OUT       M01581	// L_2nd_08 T POWER ON
; L170
LOAD      M01581	// L_2nd_08 T POWER ON
AND       T0708	// L_2nd_08 T READY 2s
OR        M0308C	// L_2nd_08 T Pos HOME >
AND NOT   T0408	// -
AND       D001140.2	// L_3rd ROT Y SVD ON
AND NOT   D002140.E	// L_3rd ROT Y ¨¬n¡íoA¢´Ao
AND NOT   M01583	// -
AND NOT   M00682	// -
AND NOT   M00683	// -
AND       M01232	// SYSTEM LEFT READY
AND       T1015	// L_P&P SS UP
AND       T4027	// L_2nd SS SPANKING BW
AND       T4029	// L_2nd SS MANDREL BW
AND       T4000	// L_1st SS TOP CLAMP    UP
AND       T4020	// L_2nd SS CLAMP.L UP
AND       T4022	// L_2nd SS CLAMP.R UP
OUT       M0308C	// L_2nd_08 T Pos HOME >
; L172
LOAD      M01583	// -
OR        M01582	// L_2nd_08 T HOME GOOD
AND NOT   M01581	// L_2nd_08 T POWER ON
AND NOT   M0308C	// L_2nd_08 T Pos HOME >
AND NOT   D002140.E	// L_3rd ROT Y ¨¬n¡íoA¢´Ao
AND NOT   M00600	// EMERGENCY ALARM
OUT       M01582	// L_2nd_08 T HOME GOOD
; L174
LOAD      D001140.8	// L_3rd ROT Y ¢¯©ªA¢®¢¯I¡¤a
OUTP      M01583	// -
; L175
LOAD      M01583	// -
OR        M01584	// -
AND       D001140.8	// L_3rd ROT Y ¢¯©ªA¢®¢¯I¡¤a
AND NOT   M03080	// L_2nd_08 T Pos.1st RECEIVE >
AND NOT   M01585	// -
OUT       M01584	// -
TON       T0408 5	// -
; L177
LOAD      T0408	// -
OR        M01585	// -
AND       T0708	// L_2nd_08 T READY 2s
AND NOT   M02081	// T)L_2nd_ 08 T JOG-
AND NOT   M02082	// T)L_2nd_ 08 T JOG+
AND       T1015	// L_P&P SS UP
AND       T4027	// L_2nd SS SPANKING BW
AND       T4029	// L_2nd SS MANDREL BW
AND       T4000	// L_1st SS TOP CLAMP    UP
AND       T4020	// L_2nd SS CLAMP.L UP
AND       T4022	// L_2nd SS CLAMP.R UP
OUT       M01585	// -
; L179
LOAD      D001140.0	// L_3rd ROT Y CTRL RDY
AND NOT   D001140.C	// L_3rd ROT Y SVD ERR
DMOV      D001142 D003880
// output comment: Read Current Position
//  Motor  OUTPUT
; L181
LOAD      F00099
OUT       D002140.0	// L_3rd ROT Y USE

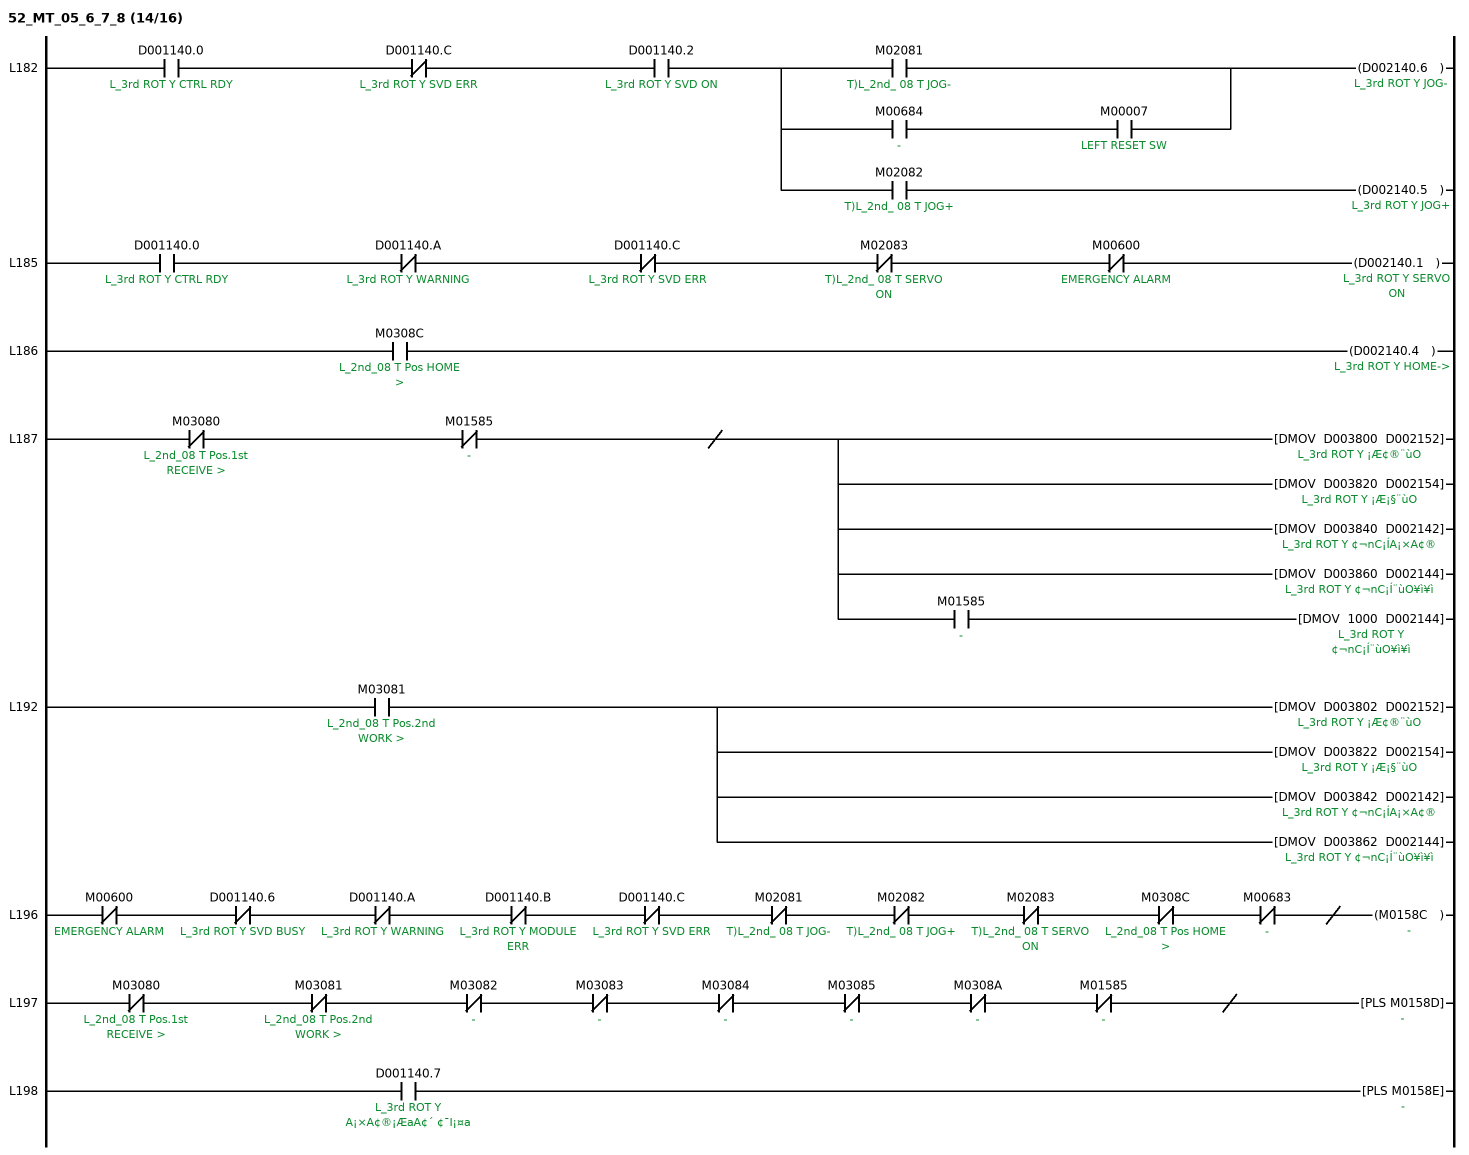
; L182
LOAD      D001140.0	// L_3rd ROT Y CTRL RDY
AND NOT   D001140.C	// L_3rd ROT Y SVD ERR
AND       D001140.2	// L_3rd ROT Y SVD ON
MPUSH
LOAD      M02081	// T)L_2nd_ 08 T JOG-
LOAD      M00684	// -
AND       M00007	// LEFT RESET SW
OR LOAD
AND LOAD
OUT       D002140.6	// L_3rd ROT Y JOG-
MPOP
AND       M02082	// T)L_2nd_ 08 T JOG+
OUT       D002140.5	// L_3rd ROT Y JOG+
; L185
LOAD      D001140.0	// L_3rd ROT Y CTRL RDY
AND NOT   D001140.A	// L_3rd ROT Y WARNING
AND NOT   D001140.C	// L_3rd ROT Y SVD ERR
AND NOT   M02083	// T)L_2nd_ 08 T SERVO ON
AND NOT   M00600	// EMERGENCY ALARM
OUT       D002140.1	// L_3rd ROT Y SERVO ON
; L186
LOAD      M0308C	// L_2nd_08 T Pos HOME >
OUT       D002140.4	// L_3rd ROT Y HOME->
; L187
LOAD NOT  M03080	// L_2nd_08 T Pos.1st RECEIVE >
AND NOT   M01585	// -
NOT
DMOV      D003800 D002152	// L_3rd ROT Y ¡Æ¢®¨ùO
DMOV      D003820 D002154	// L_3rd ROT Y ¡Æ¡§¨ùO
DMOV      D003840 D002142	// L_3rd ROT Y ¢¬nC¡ÍA¡×A¢®
DMOV      D003860 D002144	// L_3rd ROT Y ¢¬nC¡Í¨ùO¥ì¥ì
AND       M01585	// -
DMOV      1000 D002144	// L_3rd ROT Y ¢¬nC¡Í¨ùO¥ì¥ì
; L192
LOAD      M03081	// L_2nd_08 T Pos.2nd WORK >
DMOV      D003802 D002152	// L_3rd ROT Y ¡Æ¢®¨ùO
DMOV      D003822 D002154	// L_3rd ROT Y ¡Æ¡§¨ùO
DMOV      D003842 D002142	// L_3rd ROT Y ¢¬nC¡ÍA¡×A¢®
DMOV      D003862 D002144	// L_3rd ROT Y ¢¬nC¡Í¨ùO¥ì¥ì
; L196
LOAD NOT  M00600	// EMERGENCY ALARM
AND NOT   D001140.6	// L_3rd ROT Y SVD BUSY
AND NOT   D001140.A	// L_3rd ROT Y WARNING
AND NOT   D001140.B	// L_3rd ROT Y MODULE ERR
AND NOT   D001140.C	// L_3rd ROT Y SVD ERR
AND NOT   M02081	// T)L_2nd_ 08 T JOG-
AND NOT   M02082	// T)L_2nd_ 08 T JOG+
AND NOT   M02083	// T)L_2nd_ 08 T SERVO ON
AND NOT   M0308C	// L_2nd_08 T Pos HOME >
AND NOT   M00683	// -
NOT
OUT       M0158C	// -
; L197
LOAD NOT  M03080	// L_2nd_08 T Pos.1st RECEIVE >
AND NOT   M03081	// L_2nd_08 T Pos.2nd WORK >
AND NOT   M03082	// -
AND NOT   M03083	// -
AND NOT   M03084	// -
AND NOT   M03085	// -
AND NOT   M0308A	// -
AND NOT   M01585	// -
NOT
OUTP      M0158D	// -
; L198
LOAD      D001140.7	// L_3rd ROT Y A¡×A¢®¡ÆaA¢´ ¢¯I¡¤a
OUTP      M0158E	// -

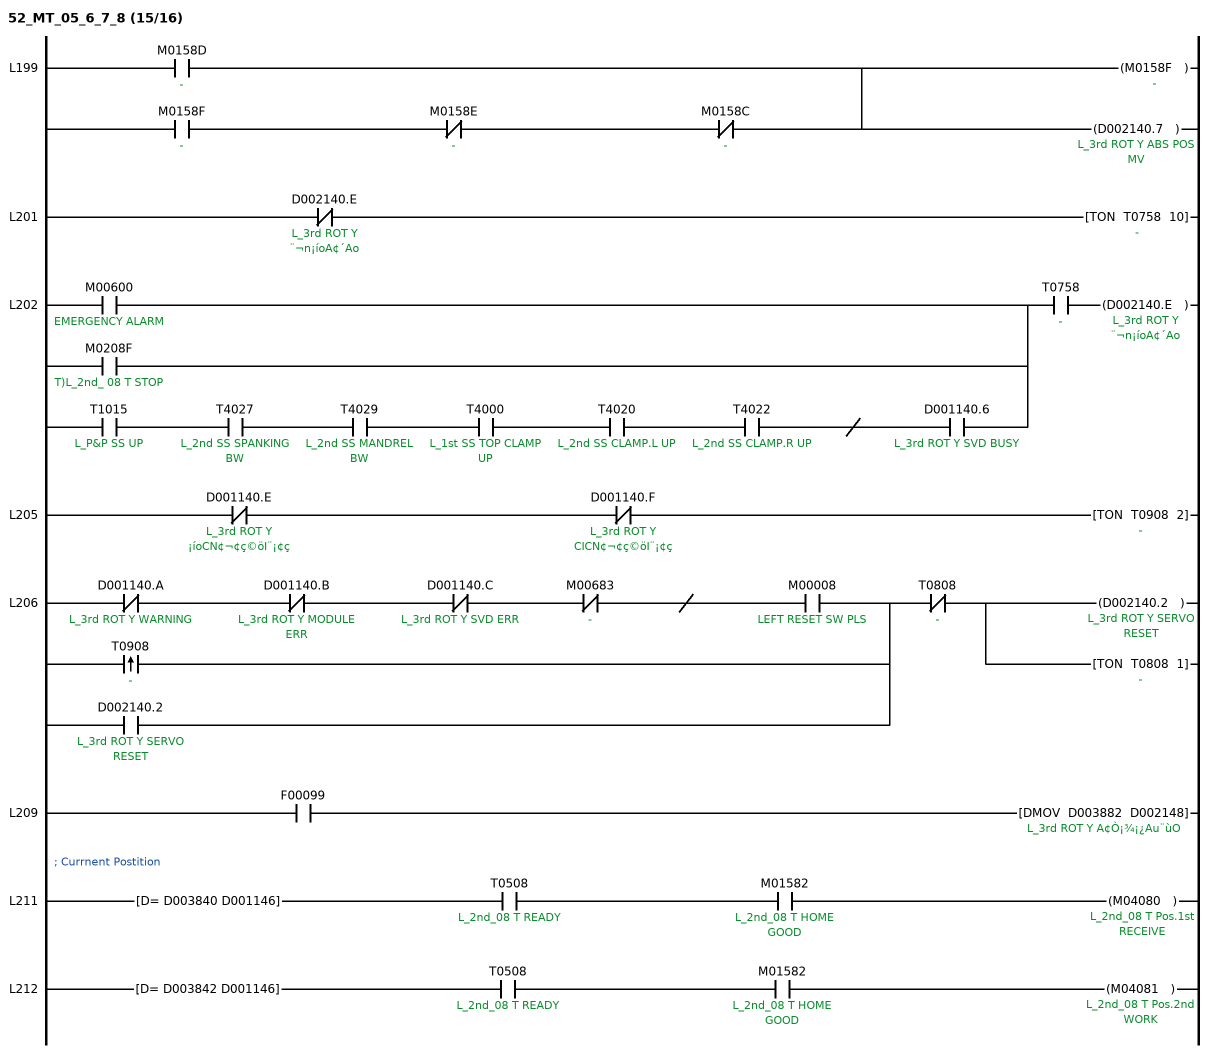
; L199
LOAD      M0158D	// -
LOAD      M0158F	// -
AND NOT   M0158E	// -
AND NOT   M0158C	// -
OR LOAD
OUT       M0158F	// -
OUT       D002140.7	// L_3rd ROT Y ABS POS MV
; L201
LOAD NOT  D002140.E	// L_3rd ROT Y ¨¬n¡íoA¢´Ao
TON       T0758 10	// -
; L202
LOAD      M00600	// EMERGENCY ALARM
OR        M0208F	// T)L_2nd_ 08 T STOP
LOAD      T1015	// L_P&P SS UP
AND       T4027	// L_2nd SS SPANKING BW
AND       T4029	// L_2nd SS MANDREL BW
AND       T4000	// L_1st SS TOP CLAMP    UP
AND       T4020	// L_2nd SS CLAMP.L UP
AND       T4022	// L_2nd SS CLAMP.R UP
NOT
AND       D001140.6	// L_3rd ROT Y SVD BUSY
OR LOAD
AND       T0758	// -
OUT       D002140.E	// L_3rd ROT Y ¨¬n¡íoA¢´Ao
; L205
LOAD NOT  D001140.E	// L_3rd ROT Y ¡íoCN¢¬¢ç©öI¨¡¢ç
AND NOT   D001140.F	// L_3rd ROT Y CICN¢¬¢ç©öI¨¡¢ç
TON       T0908 2	// -
; L206
LOAD NOT  D001140.A	// L_3rd ROT Y WARNING
AND NOT   D001140.B	// L_3rd ROT Y MODULE ERR
AND NOT   D001140.C	// L_3rd ROT Y SVD ERR
AND NOT   M00683	// -
NOT
AND       M00008	// LEFT RESET SW PLS
ORP       T0908	// -
OR        D002140.2	// L_3rd ROT Y SERVO RESET
AND NOT   T0808	// -
OUT       D002140.2	// L_3rd ROT Y SERVO RESET
TON       T0808 1	// -
; L209
LOAD      F00099
DMOV      D003882 D002148	// L_3rd ROT Y A¢Ò¡¾¡¿Au¨ùO
// Currnent Postition
; L211
LOADD=    D003840 D001146
AND       T0508	// L_2nd_08 T READY
AND       M01582	// L_2nd_08 T HOME GOOD
OUT       M04080	// L_2nd_08 T Pos.1st RECEIVE
; L212
LOADD=    D003842 D001146
AND       T0508	// L_2nd_08 T READY
AND       M01582	// L_2nd_08 T HOME GOOD
OUT       M04081	// L_2nd_08 T Pos.2nd WORK

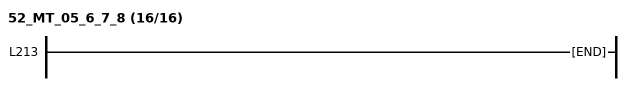
; L213
END

PROGRAM 53_MT_09_10_11_12 (task: ¨ö¨¬A¥ì CA¡¤I¡¾¡¿¡¤¡Í)

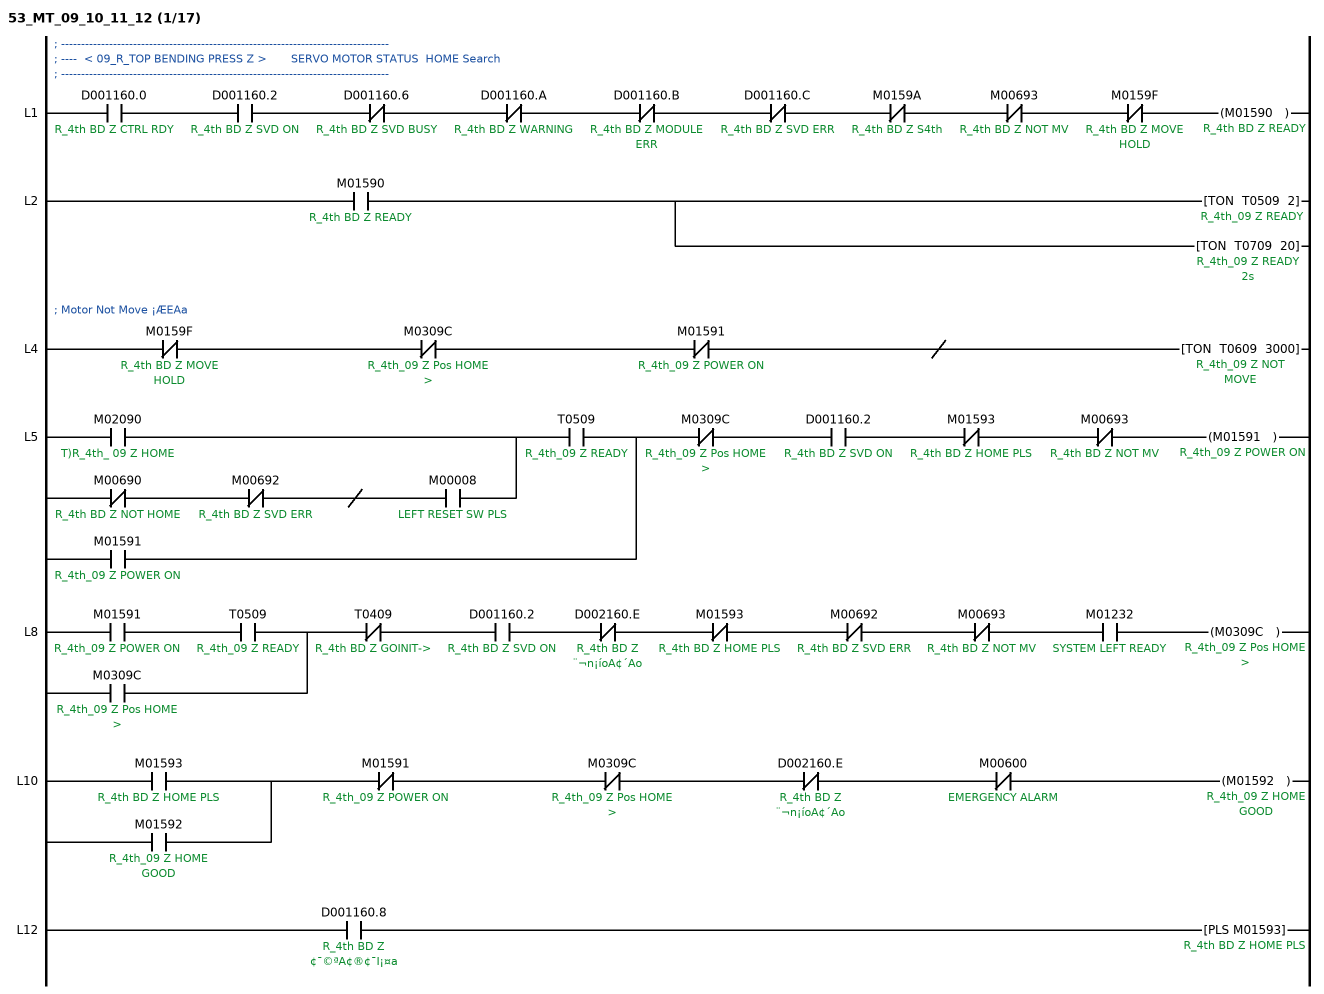
// ----------------------------------------------------------------------------------
// 
// ----  < 09_R_TOP BENDING PRESS Z >       SERVO MOTOR STATUS  HOME Search
// 
// ----------------------------------------------------------------------------------
; L1
LOAD      D001160.0	// R_4th BD Z CTRL RDY
AND       D001160.2	// R_4th BD Z SVD ON
AND NOT   D001160.6	// R_4th BD Z SVD BUSY
AND NOT   D001160.A	// R_4th BD Z WARNING
AND NOT   D001160.B	// R_4th BD Z MODULE ERR
AND NOT   D001160.C	// R_4th BD Z SVD ERR
AND NOT   M0159A	// R_4th BD Z S4th
AND NOT   M00693	// R_4th BD Z NOT MV
AND NOT   M0159F	// R_4th BD Z MOVE HOLD
OUT       M01590	// R_4th BD Z READY
; L2
LOAD      M01590	// R_4th BD Z READY
TON       T0509 2	// R_4th_09 Z READY
TON       T0709 20	// R_4th_09 Z READY 2s
; L4
LOAD NOT  M0159F	// R_4th BD Z MOVE HOLD
AND NOT   M0309C	// R_4th_09 Z Pos HOME >
AND NOT   M01591	// R_4th_09 Z POWER ON
NOT
TON       T0609 3000	// R_4th_09 Z NOT MOVE
// output comment: Motor Not Move ¡ÆEAa
; L5
LOAD      M02090	// T)R_4th_ 09 Z HOME
LOAD NOT  M00690	// R_4th BD Z NOT HOME
AND NOT   M00692	// R_4th BD Z SVD ERR
NOT
AND       M00008	// LEFT RESET SW PLS
OR LOAD
AND       T0509	// R_4th_09 Z READY
OR        M01591	// R_4th_09 Z POWER ON
AND NOT   M0309C	// R_4th_09 Z Pos HOME >
AND       D001160.2	// R_4th BD Z SVD ON
AND NOT   M01593	// R_4th BD Z HOME PLS
AND NOT   M00693	// R_4th BD Z NOT MV
OUT       M01591	// R_4th_09 Z POWER ON
; L8
LOAD      M01591	// R_4th_09 Z POWER ON
AND       T0509	// R_4th_09 Z READY
OR        M0309C	// R_4th_09 Z Pos HOME >
AND NOT   T0409	// R_4th BD Z GOINIT->
AND       D001160.2	// R_4th BD Z SVD ON
AND NOT   D002160.E	// R_4th BD Z ¨¬n¡íoA¢´Ao
AND NOT   M01593	// R_4th BD Z HOME PLS
AND NOT   M00692	// R_4th BD Z SVD ERR
AND NOT   M00693	// R_4th BD Z NOT MV
AND       M01232	// SYSTEM LEFT READY
OUT       M0309C	// R_4th_09 Z Pos HOME >
; L10
LOAD      M01593	// R_4th BD Z HOME PLS
OR        M01592	// R_4th_09 Z HOME GOOD
AND NOT   M01591	// R_4th_09 Z POWER ON
AND NOT   M0309C	// R_4th_09 Z Pos HOME >
AND NOT   D002160.E	// R_4th BD Z ¨¬n¡íoA¢´Ao
AND NOT   M00600	// EMERGENCY ALARM
OUT       M01592	// R_4th_09 Z HOME GOOD
; L12
LOAD      D001160.8	// R_4th BD Z ¢¯©ªA¢®¢¯I¡¤a
OUTP      M01593	// R_4th BD Z HOME PLS

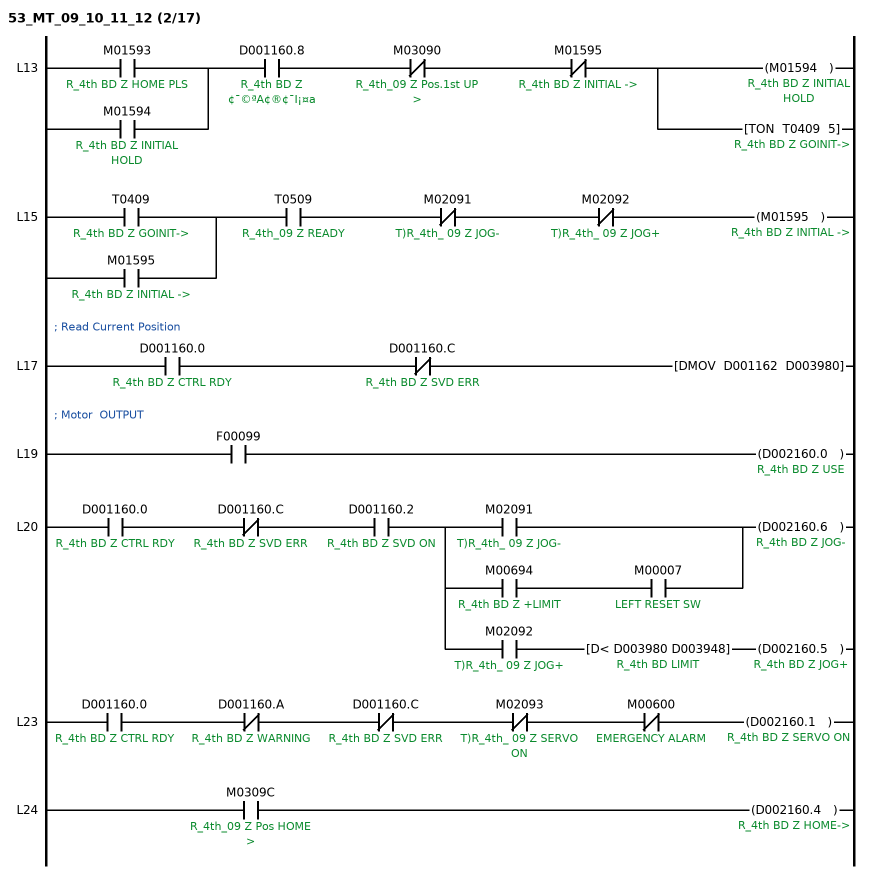
; L13
LOAD      M01593	// R_4th BD Z HOME PLS
OR        M01594	// R_4th BD Z INITIAL HOLD
AND       D001160.8	// R_4th BD Z ¢¯©ªA¢®¢¯I¡¤a
AND NOT   M03090	// R_4th_09 Z Pos.1st UP >
AND NOT   M01595	// R_4th BD Z INITIAL ->
OUT       M01594	// R_4th BD Z INITIAL HOLD
TON       T0409 5	// R_4th BD Z GOINIT->
; L15
LOAD      T0409	// R_4th BD Z GOINIT->
OR        M01595	// R_4th BD Z INITIAL ->
AND       T0509	// R_4th_09 Z READY
AND NOT   M02091	// T)R_4th_ 09 Z JOG-
AND NOT   M02092	// T)R_4th_ 09 Z JOG+
OUT       M01595	// R_4th BD Z INITIAL ->
; L17
LOAD      D001160.0	// R_4th BD Z CTRL RDY
AND NOT   D001160.C	// R_4th BD Z SVD ERR
DMOV      D001162 D003980
// output comment: Read Current Position
//  Motor  OUTPUT
; L19
LOAD      F00099
OUT       D002160.0	// R_4th BD Z USE
; L20
LOAD      D001160.0	// R_4th BD Z CTRL RDY
AND NOT   D001160.C	// R_4th BD Z SVD ERR
AND       D001160.2	// R_4th BD Z SVD ON
MPUSH
LOAD      M02091	// T)R_4th_ 09 Z JOG-
LOAD      M00694	// R_4th BD Z +LIMIT
AND       M00007	// LEFT RESET SW
OR LOAD
AND LOAD
OUT       D002160.6	// R_4th BD Z JOG-
MPOP
AND       M02092	// T)R_4th_ 09 Z JOG+
ANDD<     D003980 D003948	// R_4th BD LIMIT
OUT       D002160.5	// R_4th BD Z JOG+
; L23
LOAD      D001160.0	// R_4th BD Z CTRL RDY
AND NOT   D001160.A	// R_4th BD Z WARNING
AND NOT   D001160.C	// R_4th BD Z SVD ERR
AND NOT   M02093	// T)R_4th_ 09 Z SERVO ON
AND NOT   M00600	// EMERGENCY ALARM
OUT       D002160.1	// R_4th BD Z SERVO ON
; L24
LOAD      M0309C	// R_4th_09 Z Pos HOME >
OUT       D002160.4	// R_4th BD Z HOME->

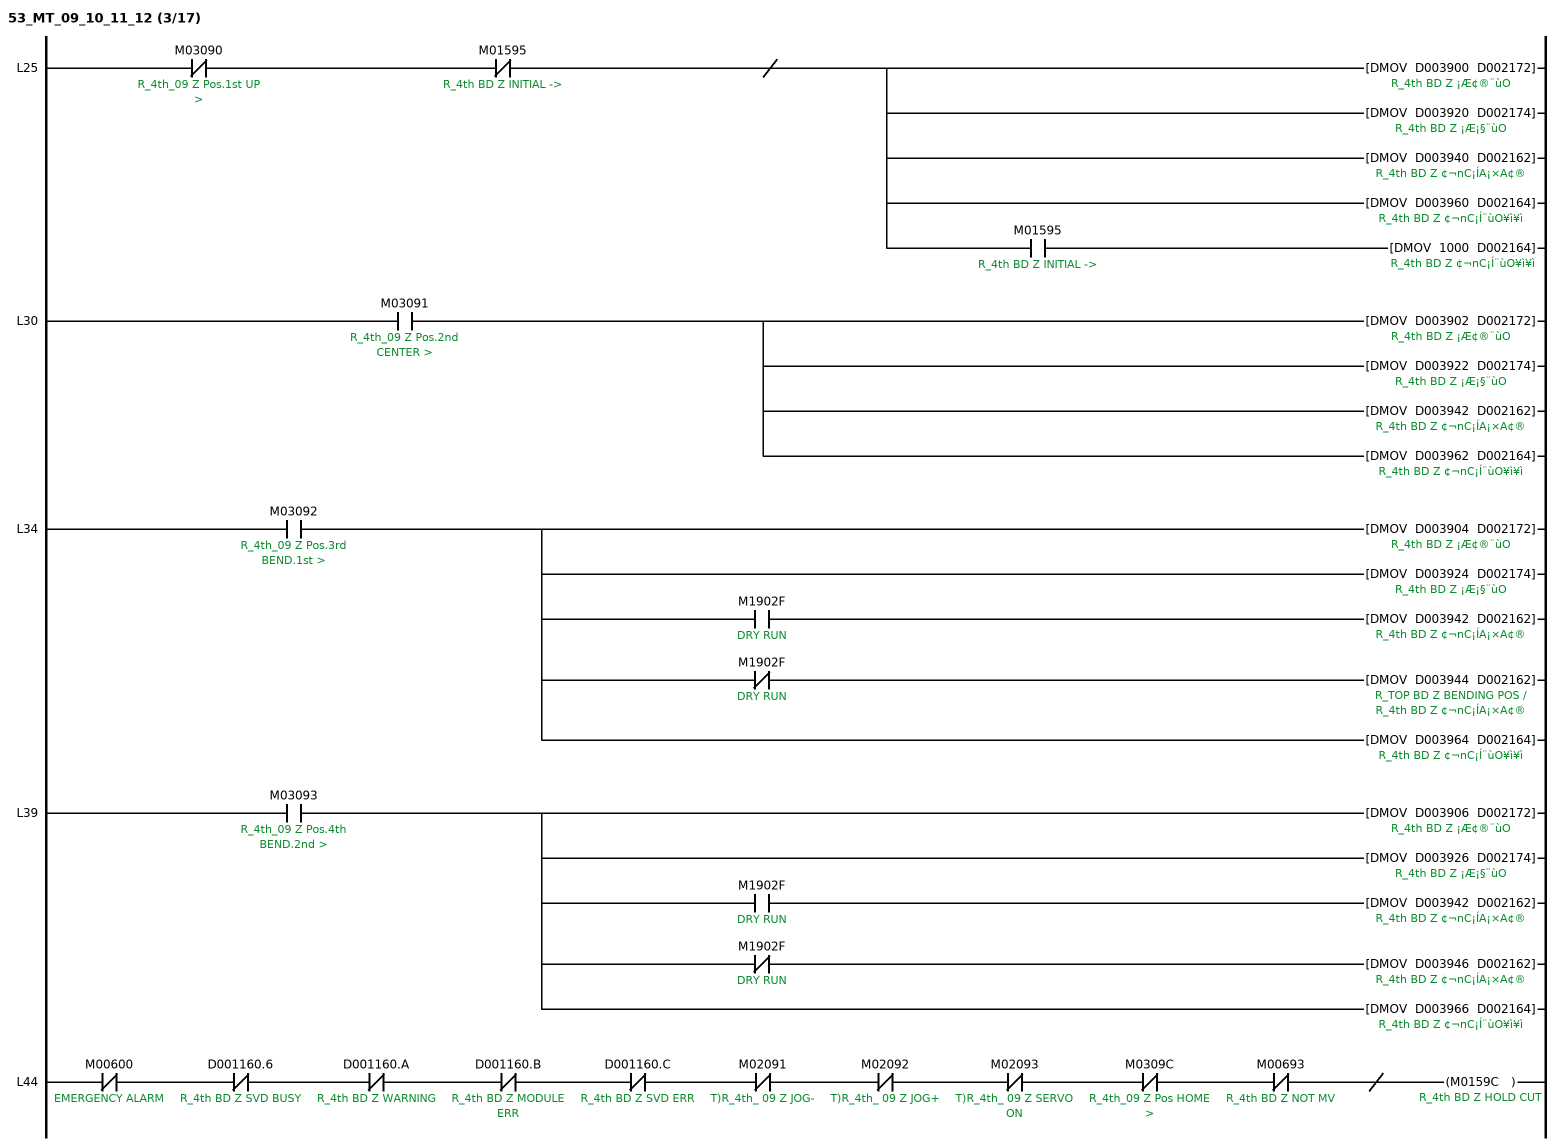
; L25
LOAD NOT  M03090	// R_4th_09 Z Pos.1st UP >
AND NOT   M01595	// R_4th BD Z INITIAL ->
NOT
DMOV      D003900 D002172	// R_4th BD Z ¡Æ¢®¨ùO
DMOV      D003920 D002174	// R_4th BD Z ¡Æ¡§¨ùO
DMOV      D003940 D002162	// R_4th BD Z ¢¬nC¡ÍA¡×A¢®
DMOV      D003960 D002164	// R_4th BD Z ¢¬nC¡Í¨ùO¥ì¥ì
AND       M01595	// R_4th BD Z INITIAL ->
DMOV      1000 D002164	// R_4th BD Z ¢¬nC¡Í¨ùO¥ì¥ì
; L30
LOAD      M03091	// R_4th_09 Z Pos.2nd CENTER >
DMOV      D003902 D002172	// R_4th BD Z ¡Æ¢®¨ùO
DMOV      D003922 D002174	// R_4th BD Z ¡Æ¡§¨ùO
DMOV      D003942 D002162	// R_4th BD Z ¢¬nC¡ÍA¡×A¢®
DMOV      D003962 D002164	// R_4th BD Z ¢¬nC¡Í¨ùO¥ì¥ì
; L34
LOAD      M03092	// R_4th_09 Z Pos.3rd BEND.1st >
DMOV      D003904 D002172	// R_4th BD Z ¡Æ¢®¨ùO
DMOV      D003924 D002174	// R_4th BD Z ¡Æ¡§¨ùO
MPUSH
AND       M1902F	// DRY RUN
DMOV      D003942 D002162	// R_4th BD Z ¢¬nC¡ÍA¡×A¢®
MLOAD
AND NOT   M1902F	// DRY RUN
DMOV      D003944 D002162	// R_TOP BD Z BENDING POS / R_4th BD Z ¢¬nC¡ÍA¡×A¢®
MPOP
DMOV      D003964 D002164	// R_4th BD Z ¢¬nC¡Í¨ùO¥ì¥ì
; L39
LOAD      M03093	// R_4th_09 Z Pos.4th BEND.2nd >
DMOV      D003906 D002172	// R_4th BD Z ¡Æ¢®¨ùO
DMOV      D003926 D002174	// R_4th BD Z ¡Æ¡§¨ùO
MPUSH
AND       M1902F	// DRY RUN
DMOV      D003942 D002162	// R_4th BD Z ¢¬nC¡ÍA¡×A¢®
MLOAD
AND NOT   M1902F	// DRY RUN
DMOV      D003946 D002162	// R_4th BD Z ¢¬nC¡ÍA¡×A¢®
MPOP
DMOV      D003966 D002164	// R_4th BD Z ¢¬nC¡Í¨ùO¥ì¥ì
; L44
LOAD NOT  M00600	// EMERGENCY ALARM
AND NOT   D001160.6	// R_4th BD Z SVD BUSY
AND NOT   D001160.A	// R_4th BD Z WARNING
AND NOT   D001160.B	// R_4th BD Z MODULE ERR
AND NOT   D001160.C	// R_4th BD Z SVD ERR
AND NOT   M02091	// T)R_4th_ 09 Z JOG-
AND NOT   M02092	// T)R_4th_ 09 Z JOG+
AND NOT   M02093	// T)R_4th_ 09 Z SERVO ON
AND NOT   M0309C	// R_4th_09 Z Pos HOME >
AND NOT   M00693	// R_4th BD Z NOT MV
NOT
OUT       M0159C	// R_4th BD Z HOLD CUT

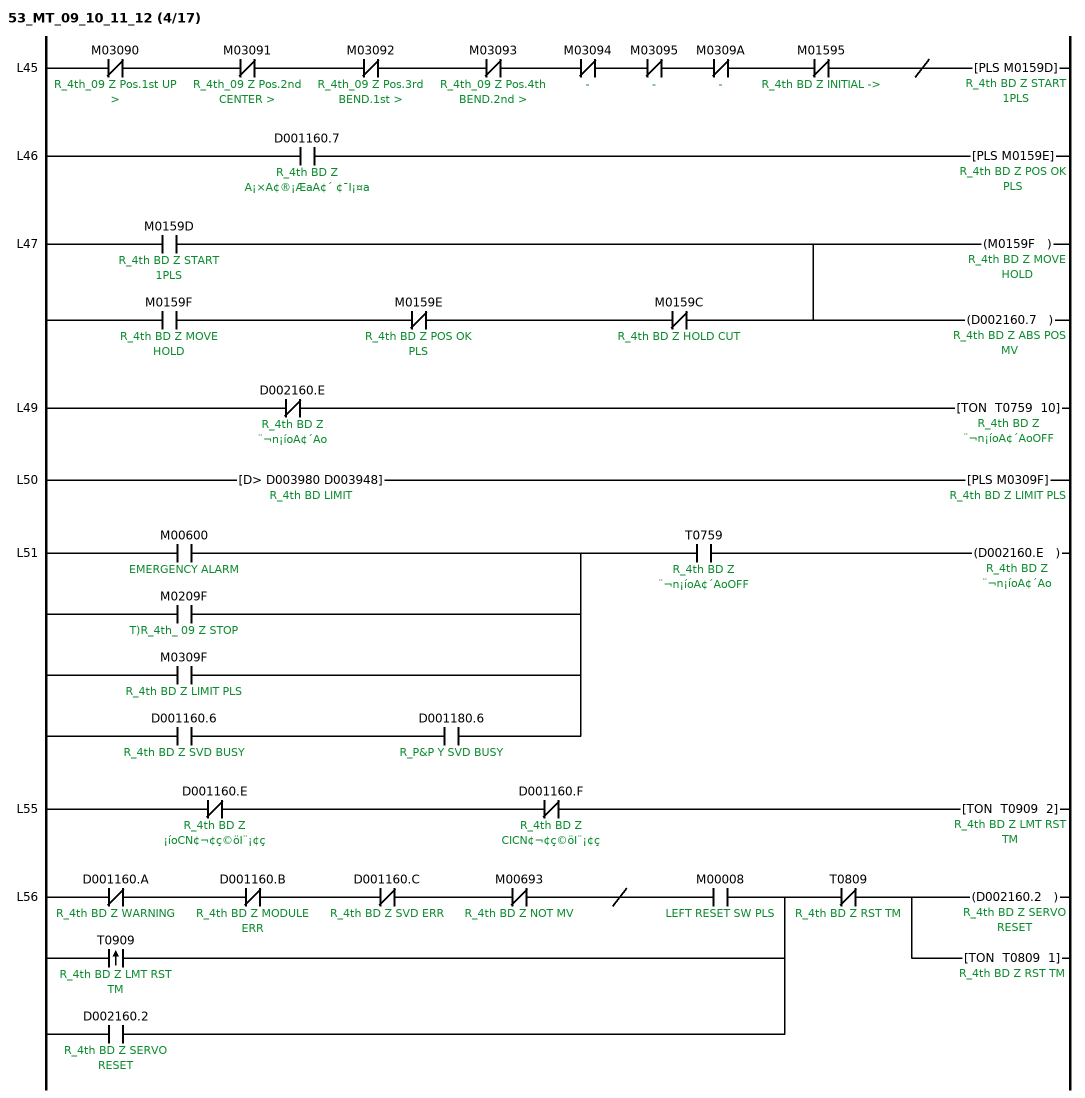
; L45
LOAD NOT  M03090	// R_4th_09 Z Pos.1st UP >
AND NOT   M03091	// R_4th_09 Z Pos.2nd CENTER >
AND NOT   M03092	// R_4th_09 Z Pos.3rd BEND.1st >
AND NOT   M03093	// R_4th_09 Z Pos.4th BEND.2nd >
AND NOT   M03094	// -
AND NOT   M03095	// -
AND NOT   M0309A	// -
AND NOT   M01595	// R_4th BD Z INITIAL ->
NOT
OUTP      M0159D	// R_4th BD Z START 1PLS
; L46
LOAD      D001160.7	// R_4th BD Z A¡×A¢®¡ÆaA¢´ ¢¯I¡¤a
OUTP      M0159E	// R_4th BD Z POS OK PLS
; L47
LOAD      M0159D	// R_4th BD Z START 1PLS
LOAD      M0159F	// R_4th BD Z MOVE HOLD
AND NOT   M0159E	// R_4th BD Z POS OK PLS
AND NOT   M0159C	// R_4th BD Z HOLD CUT
OR LOAD
OUT       M0159F	// R_4th BD Z MOVE HOLD
OUT       D002160.7	// R_4th BD Z ABS POS MV
; L49
LOAD NOT  D002160.E	// R_4th BD Z ¨¬n¡íoA¢´Ao
TON       T0759 10	// R_4th BD Z ¨¬n¡íoA¢´AoOFF
; L50
LOADD>    D003980 D003948	// R_4th BD LIMIT
OUTP      M0309F	// R_4th BD Z LIMIT PLS
; L51
LOAD      M00600	// EMERGENCY ALARM
OR        M0209F	// T)R_4th_ 09 Z STOP
OR        M0309F	// R_4th BD Z LIMIT PLS
LOAD      D001160.6	// R_4th BD Z SVD BUSY
AND       D001180.6	// R_P&P Y SVD BUSY
OR LOAD
AND       T0759	// R_4th BD Z ¨¬n¡íoA¢´AoOFF
OUT       D002160.E	// R_4th BD Z ¨¬n¡íoA¢´Ao
; L55
LOAD NOT  D001160.E	// R_4th BD Z ¡íoCN¢¬¢ç©öI¨¡¢ç
AND NOT   D001160.F	// R_4th BD Z CICN¢¬¢ç©öI¨¡¢ç
TON       T0909 2	// R_4th BD Z LMT RST TM
; L56
LOAD NOT  D001160.A	// R_4th BD Z WARNING
AND NOT   D001160.B	// R_4th BD Z MODULE ERR
AND NOT   D001160.C	// R_4th BD Z SVD ERR
AND NOT   M00693	// R_4th BD Z NOT MV
NOT
AND       M00008	// LEFT RESET SW PLS
ORP       T0909	// R_4th BD Z LMT RST TM
OR        D002160.2	// R_4th BD Z SERVO RESET
AND NOT   T0809	// R_4th BD Z RST TM
OUT       D002160.2	// R_4th BD Z SERVO RESET
TON       T0809 1	// R_4th BD Z RST TM

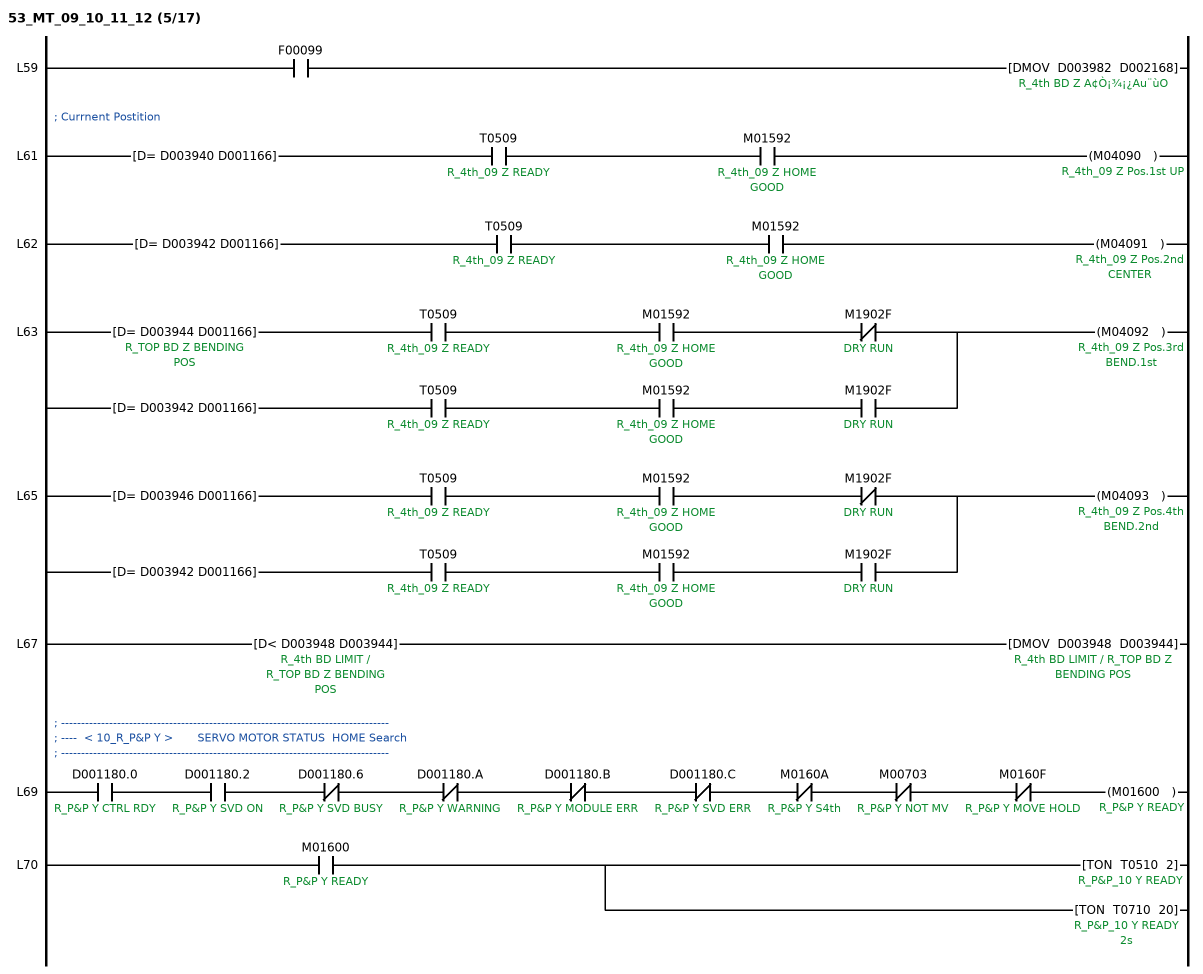
; L59
LOAD      F00099
DMOV      D003982 D002168	// R_4th BD Z A¢Ò¡¾¡¿Au¨ùO
// Currnent Postition
; L61
LOADD=    D003940 D001166
AND       T0509	// R_4th_09 Z READY
AND       M01592	// R_4th_09 Z HOME GOOD
OUT       M04090	// R_4th_09 Z Pos.1st UP
; L62
LOADD=    D003942 D001166
AND       T0509	// R_4th_09 Z READY
AND       M01592	// R_4th_09 Z HOME GOOD
OUT       M04091	// R_4th_09 Z Pos.2nd CENTER
; L63
LOADD=    D003944 D001166	// R_TOP BD Z BENDING POS
AND       T0509	// R_4th_09 Z READY
AND       M01592	// R_4th_09 Z HOME GOOD
AND NOT   M1902F	// DRY RUN
LOADD=    D003942 D001166
AND       T0509	// R_4th_09 Z READY
AND       M01592	// R_4th_09 Z HOME GOOD
AND       M1902F	// DRY RUN
OR LOAD
OUT       M04092	// R_4th_09 Z Pos.3rd BEND.1st
; L65
LOADD=    D003946 D001166
AND       T0509	// R_4th_09 Z READY
AND       M01592	// R_4th_09 Z HOME GOOD
AND NOT   M1902F	// DRY RUN
LOADD=    D003942 D001166
AND       T0509	// R_4th_09 Z READY
AND       M01592	// R_4th_09 Z HOME GOOD
AND       M1902F	// DRY RUN
OR LOAD
OUT       M04093	// R_4th_09 Z Pos.4th BEND.2nd
; L67
LOADD<    D003948 D003944	// R_4th BD LIMIT / R_TOP BD Z BENDING POS
DMOV      D003948 D003944	// R_4th BD LIMIT / R_TOP BD Z BENDING POS
// ----------------------------------------------------------------------------------
// 
// ----  < 10_R_P&P Y >       SERVO MOTOR STATUS  HOME Search
// 
// ----------------------------------------------------------------------------------
; L69
LOAD      D001180.0	// R_P&P Y CTRL RDY
AND       D001180.2	// R_P&P Y SVD ON
AND NOT   D001180.6	// R_P&P Y SVD BUSY
AND NOT   D001180.A	// R_P&P Y WARNING
AND NOT   D001180.B	// R_P&P Y MODULE ERR
AND NOT   D001180.C	// R_P&P Y SVD ERR
AND NOT   M0160A	// R_P&P Y S4th
AND NOT   M00703	// R_P&P Y NOT MV
AND NOT   M0160F	// R_P&P Y MOVE HOLD
OUT       M01600	// R_P&P Y READY
; L70
LOAD      M01600	// R_P&P Y READY
TON       T0510 2	// R_P&P_10 Y READY
TON       T0710 20	// R_P&P_10 Y READY 2s

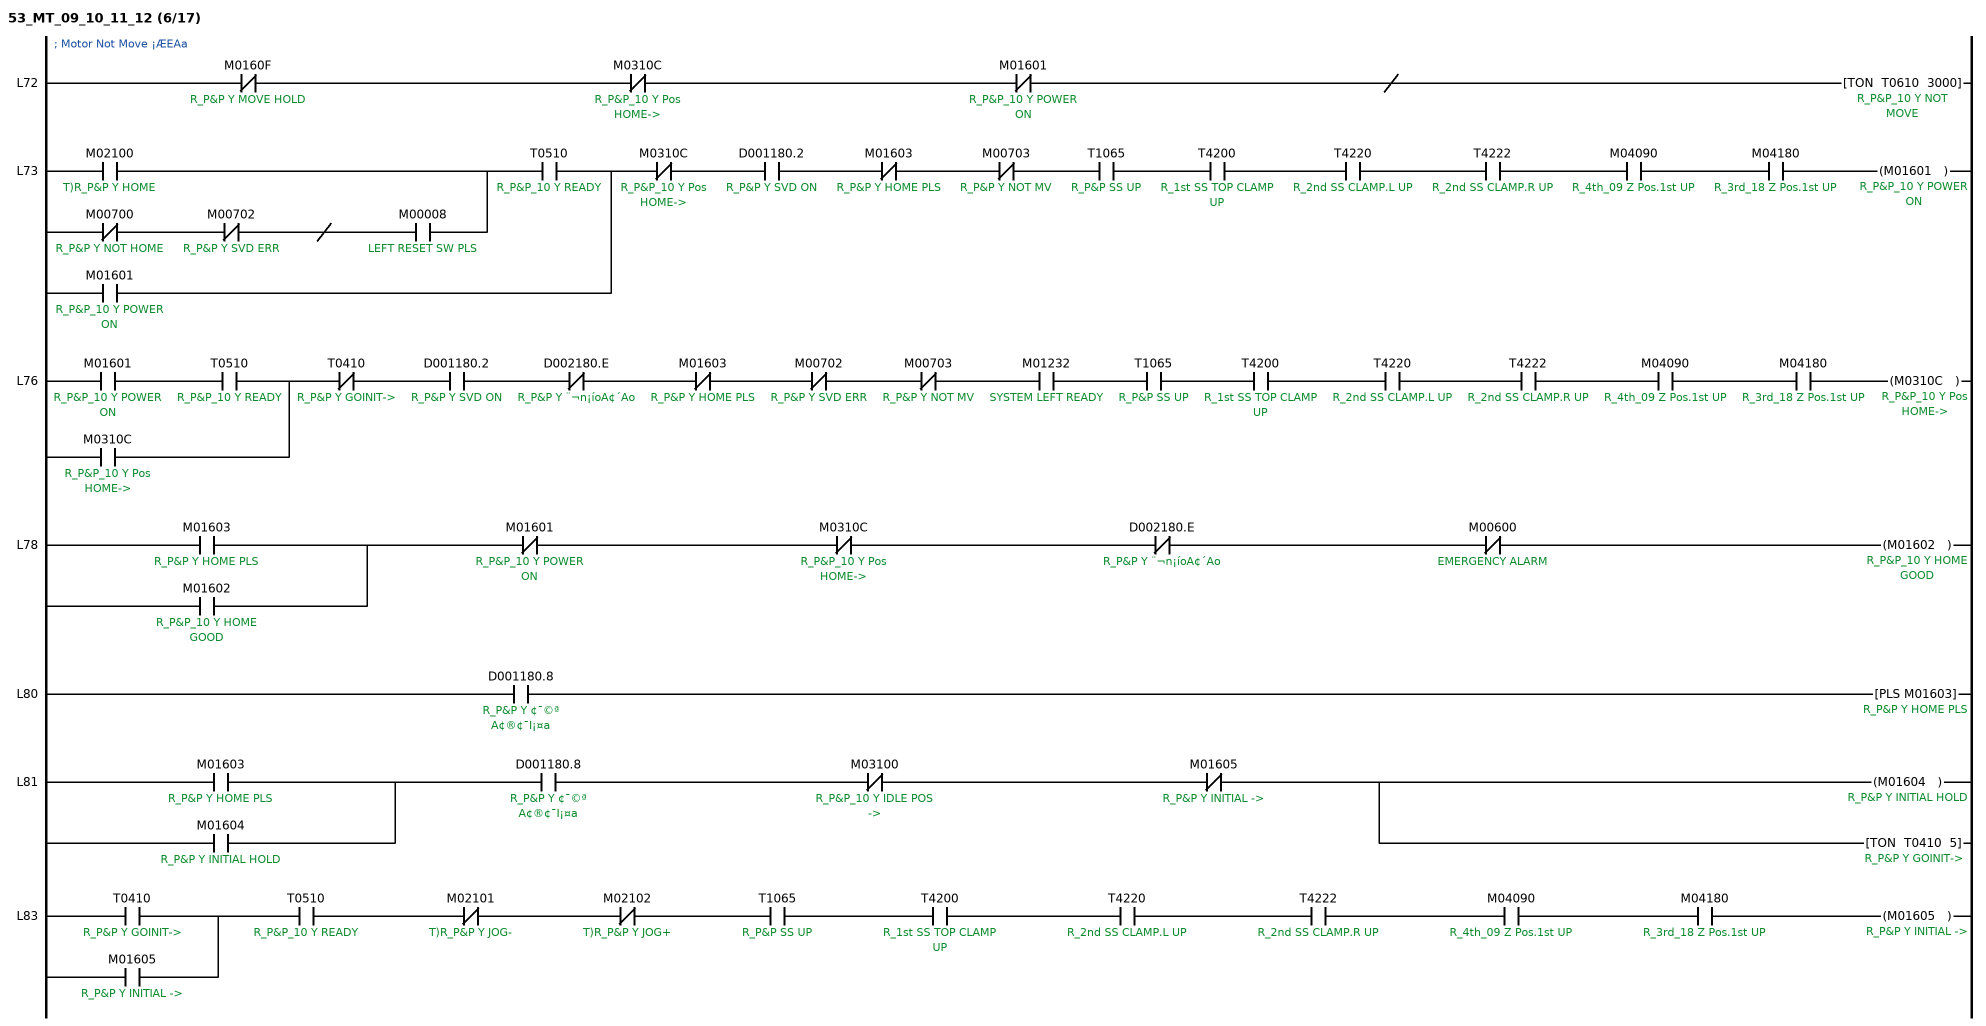
; L72
LOAD NOT  M0160F	// R_P&P Y MOVE HOLD
AND NOT   M0310C	// R_P&P_10 Y Pos HOME->
AND NOT   M01601	// R_P&P_10 Y POWER ON
NOT
TON       T0610 3000	// R_P&P_10 Y NOT MOVE
// output comment: Motor Not Move ¡ÆEAa
; L73
LOAD      M02100	// T)R_P&P Y HOME
LOAD NOT  M00700	// R_P&P Y NOT HOME
AND NOT   M00702	// R_P&P Y SVD ERR
NOT
AND       M00008	// LEFT RESET SW PLS
OR LOAD
AND       T0510	// R_P&P_10 Y READY
OR        M01601	// R_P&P_10 Y POWER ON
AND NOT   M0310C	// R_P&P_10 Y Pos HOME->
AND       D001180.2	// R_P&P Y SVD ON
AND NOT   M01603	// R_P&P Y HOME PLS
AND NOT   M00703	// R_P&P Y NOT MV
AND       T1065	// R_P&P SS UP
AND       T4200	// R_1st SS TOP CLAMP UP
AND       T4220	// R_2nd SS CLAMP.L UP
AND       T4222	// R_2nd SS CLAMP.R UP
AND       M04090	// R_4th_09 Z Pos.1st UP
AND       M04180	// R_3rd_18 Z Pos.1st UP
OUT       M01601	// R_P&P_10 Y POWER ON
; L76
LOAD      M01601	// R_P&P_10 Y POWER ON
AND       T0510	// R_P&P_10 Y READY
OR        M0310C	// R_P&P_10 Y Pos HOME->
AND NOT   T0410	// R_P&P Y GOINIT->
AND       D001180.2	// R_P&P Y SVD ON
AND NOT   D002180.E	// R_P&P Y ¨¬n¡íoA¢´Ao
AND NOT   M01603	// R_P&P Y HOME PLS
AND NOT   M00702	// R_P&P Y SVD ERR
AND NOT   M00703	// R_P&P Y NOT MV
AND       M01232	// SYSTEM LEFT READY
AND       T1065	// R_P&P SS UP
AND       T4200	// R_1st SS TOP CLAMP UP
AND       T4220	// R_2nd SS CLAMP.L UP
AND       T4222	// R_2nd SS CLAMP.R UP
AND       M04090	// R_4th_09 Z Pos.1st UP
AND       M04180	// R_3rd_18 Z Pos.1st UP
OUT       M0310C	// R_P&P_10 Y Pos HOME->
; L78
LOAD      M01603	// R_P&P Y HOME PLS
OR        M01602	// R_P&P_10 Y HOME GOOD
AND NOT   M01601	// R_P&P_10 Y POWER ON
AND NOT   M0310C	// R_P&P_10 Y Pos HOME->
AND NOT   D002180.E	// R_P&P Y ¨¬n¡íoA¢´Ao
AND NOT   M00600	// EMERGENCY ALARM
OUT       M01602	// R_P&P_10 Y HOME GOOD
; L80
LOAD      D001180.8	// R_P&P Y ¢¯©ªA¢®¢¯I¡¤a
OUTP      M01603	// R_P&P Y HOME PLS
; L81
LOAD      M01603	// R_P&P Y HOME PLS
OR        M01604	// R_P&P Y INITIAL HOLD
AND       D001180.8	// R_P&P Y ¢¯©ªA¢®¢¯I¡¤a
AND NOT   M03100	// R_P&P_10 Y IDLE POS ->
AND NOT   M01605	// R_P&P Y INITIAL ->
OUT       M01604	// R_P&P Y INITIAL HOLD
TON       T0410 5	// R_P&P Y GOINIT->
; L83
LOAD      T0410	// R_P&P Y GOINIT->
OR        M01605	// R_P&P Y INITIAL ->
AND       T0510	// R_P&P_10 Y READY
AND NOT   M02101	// T)R_P&P Y JOG-
AND NOT   M02102	// T)R_P&P Y JOG+
AND       T1065	// R_P&P SS UP
AND       T4200	// R_1st SS TOP CLAMP UP
AND       T4220	// R_2nd SS CLAMP.L UP
AND       T4222	// R_2nd SS CLAMP.R UP
AND       M04090	// R_4th_09 Z Pos.1st UP
AND       M04180	// R_3rd_18 Z Pos.1st UP
OUT       M01605	// R_P&P Y INITIAL ->

